(* CODESYS project lcls-twincat-motion-v1.3.3 (1).library
   Company: SLAC
   Title: lcls-twincat-motion
   Placeholder: lcls-twincat-motion
   Version: 1.3.3

Project tree, tasks and I/O mapping:
  libraries: LCLS General, * (SLAC); PMPS, * (SLAC - LCLS); Tc2_EtherCAT, * (Beckhoff Automation GmbH); Tc2_MC2, * (Beckhoff Automation GmbH); Tc2_Standard, * (Beckhoff Automation GmbH); Tc2_System, * (Beckhoff Automation GmbH); Tc2_Utilities, * (Beckhoff Automation GmbH); Tc3_Module, * (Beckhoff Automation GmbH)
  DUTs/
    data type DUT_MotionPneumaticActuator
    data type DUT_MotionStage
    data type DUT_PositionState
    data type EL5042_Status
    data type ENUM_EpicsHomeCmd
    data type ENUM_EpicsInOut
    data type ENUM_EpicsMotorCmd
    data type ENUM_MotionRequest
    data type ENUM_PnuematicActuatorPositionState
    data type ENUM_StageBrakeMode
    data type ENUM_StageEnableMode
    data type ST_RenishawAbsEnc
  GVLs/
    global variables MOTION_GVL
  POUs/
    Deprecated/
      function block FB_EpicsInOut [ST]
      function block FB_PositionStateManager [ST]
      function block FB_StatePTPMove [ST]
    ImplicitChecks/
      function CheckBounds [ST]
      function CheckDivDInt [ST]
      function CheckDivLInt [ST]
      function CheckDivLReal [ST]
      function CheckDivReal [ST]
    Motion/
      Gantry/
        function block FB_GantryAutoCoupling [ST]
        function block FB_GantryDiffVirtualLimitSwitch [ST]
      PMPS/
        function block FB_EncErrorFFO [ST]
        function block FB_NCErrorFFO [ST]
        function block FB_PositionStatePMPS [ST]: AssertHere, ClearAsserts, HandleBPTM, HandleFFO
        function block FB_PositionStatePMPS_Base [ST]: AssertHere, ClearAsserts, Exec, GetBeamFromState, GetStateCode, GetStateStruct, HandleBPTM, HandleFFO
        function block FB_PositionStatePMPS_Test [ST]: HandleBPTM, HandleFFO
      States/
        Examples/
          function block FB_PositionStateInOut [ST]
          function block FB_PositionStateInOut_WithPMPS [ST]
          function block FB_PositionStateInOut_WithPMPS_Test [ST]
        Helpers/
          function F_AtPositionState [ST]
          function F_PosOverLowerBound [ST]
          function F_PosUnderUpperBound [ST]
          function F_PosWithinDelta [ST]
          function block FB_RawCountConverter [ST]
        Internals/
          function block FB_PositionStateInternal [ST]
          function block FB_PositionStateLock [ST]
        function block FB_PositionStateBase [ST]: Exec, StateHandler
        function block FB_PositionStateBase_WithPMPS [ST]: Exec, PMPSHandler
        function block FB_PositionStateBase_WithPMPS_Test [ST]: Exec, PMPSHandler
        function block FB_PositionStateMove [ST]
      Utils/
        function F_MotionErrorCodeLookup [ST]
        function block FB_SetEnables [ST]
      function block FB_EncoderValue [ST]
      function block FB_MotionPneumaticActuator [ST]: ACT_IO, ACT_Logger
      function block FB_MotionRequest [ST]
      function block FB_MotionStage [ST]
      function block FB_MotionStageNCParams [ST]
      function block FB_MotionStageSim [ST]
    MotorTesting/
      function block FB_MicroStepCountTest [ST]
  tc_mca_std_lib/
    DUTs/
      data type DUT_AxisStatus_v0_01
    GVLs/
      global variables GVL
    POUs/
      ChangeConfig/
        function block FB_ReadFloatParameter [ST]
        function block FB_ReadParameterInNc_v1_00 [ST]
        function block FB_WriteFloatParameter [ST]
        function block FB_WriteParameterInNc_v1_00 [ST]
      ErrorHandling/
        data type DUT_ErrorState
        data type DUT_TerminalError
        function block FB_ErrorList [ST]
        function block FB_TerminalError [ST]
        global variables GVL_ErrorSystem
        data type ST_ErrorSystem
      Hardware/
        EtherCAT_Terminals/
          Analog_Inputs/
            function block EL3174_0002 [ST]
            function block EL3214 [ST]
            function block EL3255 [ST]
            function block FB_CalculateFrequency_3702_v0_01 [ST]
          Digital_Inputs/
            function block EL1008 [ST]
            function block EL1018 [ST]
            function block EL1808 [ST]
            function block EL1809 [ST]
            function block EL1819 [ST]
            function block FB_EL1252ASM_v1_00 [ST]
          Digital_Outputs/
            External_Types/
              data type dutEL2521_Ctrl
              data type dutEL2521_Status
            function block EL2014 [ST]
            function block EL2252 [ST]
            function block EL2808 [ST]
            function block EL2819 [ST]
          Measuring_Terminals/
            function block EL5002 [ST]
            function block EL5021 [ST]
            function block EL5042 [ST]
            function block EL5101 [ST]
          Motion/
            function block EL7211_v1_00 [ST]
            function block EL9576_v1_00 [ST]
          System/
            function block EL9410 [ST]
            function block EL9505 [ST]
        Other/
          function block EK1200 [ST]
      Motion/
        Homing/
          function block FB_HomeDirect [ST]
          function block FB_HomeFinish [ST]
          function block FB_HomePrepare [ST]
          function block FB_HomeReadNcVelocities [ST]
          function block FB_HomeReadSoftLimEnable [ST]
          function block FB_HomeToSwitch [ST]
          function block FB_HomeVirtual [ST]
          function block FB_HomeWriteNcVelocities [ST]
          function block FB_HomeWriteSoftLimEnable [ST]
        function block FB_DriveVirtual [ST]
        function block FB_NcAxis [ST]
  UnitTests/
    program BasicTests [ST]
    program Interactive [ST]
  Version/
    global variables Global_Version
*)

// DUTs/DUT_MotionPneumaticActuator
{attribute 'qualified_only'}
{attribute 'strict'}
TYPE DUT_MotionPneumaticActuator :
    // Defines the EPICS interface to actuating a pneumatic stage
STRUCT
     (* Hardware *)
    //Readbacks
    //Limit Switch
    {attribute 'pytmc' := '
     pv: PLC:bInLimitSwitch
     io: i
     field: ZNAM FALSE
     field: ONAM TRUE
     field: DESC TRUE if IN limit is reached
    '}
    i_bInLimitSwitch    :    BOOL;
    {attribute 'pytmc' := '
     pv: PLC:bOutLimitSwitch
     io: i
     field: ZNAM FALSE
     field: ONAM TRUE
     field: DESC TRUE if OUT limit is reached
    '}
    i_bOutLimitSwitch    :    BOOL;
    //Controls
    //Digital outputs
    {attribute 'pytmc' := '
    pv: bRetractDigitalOutput;
    io: i;
    field: ONAM FALSE
    field: ZNAM TRUE
    field: DESC TRUE if Retract digital output is active
    '}
    q_bRetract    :    BOOL;
    {attribute 'pytmc' := '
    pv: bInsetDigitalOutput;
    io: i;
    field: ONAM FALSE
    field: ZNAM TRUE
    field: DESC TRUE if Insert digital output is active
    '}
    q_bInsert    :    BOOL;


    //Logic and supervisory
    {attribute 'pytmc' := '
    pv: bInterlockOK;
    io: i;
    field: ZNAM FALSE
    field: ONAM TRUE
    field: DESC True if the actuator has permission to move in either direction
    '}
    bILK_OK: BOOL;
    {attribute 'pytmc' := '
    pv: bInsertEnable;
    io: i;
    field: ZNAM FALSE
    field: ONAM TRUE
    field: DESC True if the actuator had permission to be retracted
    '}
    bInsertOK    :    BOOL;
    {attribute 'pytmc' := '
    pv: bRetractEnable;
    io: i;
    field: ZNAM FALSE
    field: ONAM TRUE
    field: DESC True if the actuator had permission to be inserted
    '}
    bRetractOK    :    BOOL;

    (* Commands *)
    // Used from Epics to comand the actuator to  move
    {attribute 'pytmc' := '
    pv: CMD:IN;
    io: io;
    field: DESC Used by EPICS and internally to request Insert motion
    '}
    bInsert_SW        :    BOOL;
    {attribute 'pytmc' := '
    pv: CMD:OUT;
    io: io;
    field: DESC Used by EPICS and internally to request retract motion
    '}
    bRetract_SW    :    BOOL;

    (*Returns*)
     // TRUE if in the middle of a command
    {attribute 'pytmc' := '
     pv: bBusy
     io: i
     field: ONAM FALSE
     field: ZNAM TRUE
     field: DESC TRUE if in the middle of a command
    '}
    bBusy: BOOL;
    // TRUE if we've done a command and it has finished
    {attribute 'pytmc' := '
     pv: bDone
     io: i
     field: ONAM FALSE
     field: ZNAM TRUE
      field: DESC TRUE if command finished successfully
    '}
    bDone: BOOL;
     {attribute 'pytmc' := '
        pv: bReset
        io: io
        field: ZNAM FALSE
        field: ONAM TRUE
        field: DESC Used internally to reset errors
    '}
    bReset: BOOL;
    // TRUE if we're in an error state
    {attribute 'pytmc' := '
     pv: PLC:bError
     io: i
     field: ONAM FALSE
     field: ZNAM TRUE
     field: DESC TRUE if we're in an error state
    '}
    bError: BOOL;

     // Error code if nonzero
    {attribute 'pytmc' := '
     pv: PLC:nErrorId
     io: i
     field: DESC Error code if nonzero
    '}
    nErrorId: UDINT;
    // Message to identify the error state
    {attribute 'pytmc' := '
     pv: PLC:sErrorMessage
     io: i
     field: DESC Message to identify the error state
    '}
    sErrorMessage: STRING;
    {attribute 'pytmc' := '
    pv: nPositionState ;
    type: mbbi ;
    field: ZRST RETRACTED ;
    field: ONST INSERTED ;
    field: TWST MOVING ;
    field: THST INVALID ;
    io: i
    field: DESC Pneumatic actuator position
    '}

    eState    :    ENUM_PnuematicActuatorPositionState := ENUM_PnuematicActuatorPositionState.INVALID;

END_STRUCT
END_TYPE

// DUTs/DUT_MotionStage
TYPE DUT_MotionStage :
    // Defines the EPICS interface to moving a motor in TwinCAT
STRUCT
    (* Hardware *)

    // PLC Axis Reference
    Axis: AXIS_REF;
    // NC Forward Limit Switch: TRUE if ok to move
    {attribute 'pytmc' := '
        pv: PLC:bLimitForwardEnable
        io: i
        field: ZNAM FALSE
        field: ONAM TRUE
        field: DESC FALSE if forward limit hit
    '}
    bLimitForwardEnable AT %I*: BOOL;
    // NC Backward Limit Switch: TRUE if ok to move
    {attribute 'pytmc' := '
        pv: PLC:bLimitBackwardEnable
        io: i
        field: ZNAM FALSE
        field: ONAM TRUE
        field: DESC FALSE if reverse limit hit
    '}
    bLimitBackwardEnable AT %I*: BOOL;
    // NO Home Switch: TRUE if at home
    {attribute 'pytmc' := '
        pv: PLC:bHome
        io: i
        field: ZNAM FALSE
        field: ONAM TRUE
        field: DESC TRUE if at homing switch
    '}
    bHome AT %I*: BOOL;
    // NC Brake Output: TRUE to release brake
    {attribute 'pytmc' := '
        pv: PLC:bBrakeRelease
        io: i
        field: ZNAM FALSE
        field: ONAM TRUE
        field: DESC TRUE if brake released
    '}
    bBrakeRelease AT %Q*: BOOL;
    // NC STO Input: TRUE if ok to move
    {attribute 'pytmc' := '
        pv: PLC:bHardwareEnable
        io: i
        field: ZNAM FALSE
        field: ONAM TRUE
        field: DESC TRUE if STO not hit
    '}
    bHardwareEnable AT %I*: BOOL;

    // Raw encoder IO for ULINT (Biss-C)
    nRawEncoderULINT AT %I*: ULINT;
    // Raw encoder IO for UINT (Relative Encoders)
    nRawEncoderUINT AT %I*: UINT;
    // Raw encoder IO for INT (LVDT)
    nRawEncoderINT AT %I*: INT;

    (* Psuedo-hardware *)

    // Forward enable EPS summary
    {attribute 'pytmc' := '
        pv: PLC:bAllForwardEnable
        io: i
        field: ZNAM FALSE
        field: ONAM TRUE
        field: DESC Summary of axis permission to move forward
    '}
    bAllForwardEnable: BOOL:=FALSE;
    // Backward enable EPS summary
    {attribute 'pytmc' := '
        pv: PLC:bAllBackwardEnable
        io: i
        field: ZNAM FALSE
        field: ONAM TRUE
        field: DESC Summary of axis permission to move backward
    '}
    bAllBackwardEnable: BOOL:=FALSE;
    // Enable EPS summary encapsulating emergency stop button and any additional motion preventive hardware
    {attribute 'pytmc' := '
        pv: PLC:bAllEnable
        io: i
        field: ZNAM FALSE
        field: ONAM TRUE
        field: DESC Summary of axis permission to have power
    '}
    bAllEnable: BOOL:=FALSE;
    // Forward virtual gantry limit switch
    {attribute 'pytmc' := '
        pv: PLC:bGantryForwardEnable
        io: i
        field: ZNAM FALSE
        field: ONAM TRUE
        field: DESC TRUE if gantry ok to move forward
    '}
    bGantryForwardEnable: BOOL:=FALSE;
    // Backward virtual gantry limit switch
    {attribute 'pytmc' := '
        pv: PLC:bGantryBackwardEnable
        io: i
        field: ZNAM FALSE
        field: ONAM TRUE
        field: DESC TRUE if gantry ok to move backward
    '}
    bGantryBackwardEnable: BOOL:=FALSE;
    // Encoder count summary, if linked above
    {attribute 'pytmc' := '
        pv: PLC:nEncoderCount
        io: i
        field: DESC Count from encoder hardware
    '}
    nEncoderCount: UDINT;

    (* Settings *)
    // Name to use for log messages, fast faults, etc.
    {attribute 'pytmc' := '
        pv: PLC:sName
        io: i
        field: DESC PLC program name
    '}
    sName: STRING;
    // If TRUE, we want to enable the motor independently of PMPS or other safety systems.
    {attribute 'pytmc' := '
        pv: PLC:bPowerSelf
        io: i
        field: ZNAM FALSE
        field: ONAM TRUE
        field: DESC FALSE if axis is in PMPS
    '}
    bPowerSelf: BOOL:=FALSE;
    // Determines when we automatically enable the motor
    {attribute 'pytmc' := '
        pv: PLC:nEnableMode
        io: i
        field: DESC Describes when the axis will automatically get power
    '}
    nEnableMode: ENUM_StageEnableMode:=ENUM_StageEnableMode.DURING_MOTION;
    // Determines when we automatically disengage the brake
    {attribute 'pytmc' := '
        pv: PLC:nBrakeMode
        io: i
        field: DESC Describes when the brake will be released
    '}
    nBrakeMode: ENUM_StageBrakeMode:=ENUM_StageBrakeMode.IF_ENABLED;
    // Determines our encoder homing strategy
    {attribute 'pytmc' := '
        pv: PLC:nHomingMode
        io: i
        field: DESC Describes our homing strategy
    '}
    nHomingMode: ENUM_EpicsHomeCmd:=ENUM_EpicsHomeCmd.NONE;
    // Set true to activate gantry EPS
    {attribute 'pytmc' := '
        pv: PLC:bGantryAxis
        io: i
        field: ZNAM FALSE
        field: ONAM TRUE
        field: DESC TRUE if gantry EPS active
    '}
    bGantryAxis: BOOL:=FALSE;

    // Set to gantry difference tolerance
    nGantryTol: LINT:=0;

    // Encoder count at which this axis is aligned with other axis
    nEncRef: ULINT:=0;

    (* Commands *)
    // Used internally to request enables
    {attribute 'pytmc' := '
        pv: PLC:bEnable
        io: io
        field: ZNAM FALSE
        field: ONAM TRUE
        field: DESC Used internally to request enables
    '}
    bEnable: BOOL;
    // Used internally to reset errors and other state
    {attribute 'pytmc' := '
        pv: PLC:bReset
        io: io
        field: ZNAM FALSE
        field: ONAM TRUE
        field: DESC Used internally to reset errors
    '}
    bReset: BOOL;
    // Used internally and by the IOC to start or stop a move
    {attribute 'pytmc' := '
        pv: PLC:bExecute
        io: io
        field: ZNAM FALSE
        field: ONAM TRUE
        field: DESC Used internally and by the IOC to start or stop
    '}
    bExecute: BOOL;

    (* Command Args *)
    // Used internally and by the IOC to pick what kind of move to do
    {attribute 'pytmc' := '
        pv: PLC:nCommand
        io: io
        field: DESC Used internally and by the IOC to pick move type
    '}
    nCommand: INT;
    // Used internally and by the IOC to pass additional data to some commands
    {attribute 'pytmc' := '
        pv: PLC:nCmdData
        io: io
        field: DESC Used internally and by the IOC to pass extra args
    '}
    nCmdData: INT;
    // Used internally and by the IOC to pick a destination for the move
    {attribute 'pytmc' := '
        pv: PLC:fPosition
        io: io
        field: DESC Used internally and by the IOC as the set position
    '}
    fPosition: LREAL;
    // Used internally and by the IOC to pick a move velocity
    {attribute 'pytmc' := '
        pv: PLC:fVelocity
        io: io
        field: DESC Used internally and by the IOC to set velocity
    '}
    fVelocity: LREAL;
    // Used internally and by the IOC to pick a move acceleration
    {attribute 'pytmc' := '
        pv: PLC:fAcceleration
        io: io
        field: DESC Used internally and by the IOC to set acceleration
    '}
    fAcceleration: LREAL;
    // Used internally and by the IOC to pick a move deceleration
    {attribute 'pytmc' := '
        pv: PLC:fDeceleration
        io: io
        field: DESC Used internally and by the IOC to set deceleration
    '}
    fDeceleration: LREAL;
    // Used internally and by the IOC to pick a home position
    {attribute 'pytmc' := '
        pv: PLC:fHomePosition
        io: io
        field: DESC Used internally and by the IOC to pick home position
    '}
    fHomePosition: LREAL;

    (* Info *)
    // Unique ID assigned to each axis in the NC
    {attribute 'pytmc' := '
        pv: PLC:nMotionAxisID
        io: i
        field: DESC Unique ID assigned to each axis in the NC
    '}
    nMotionAxisID: UDINT:=0;

    (* Returns *)
    // TRUE if done enabling
    {attribute 'pytmc' := '
        pv: PLC:bEnableDone
        io: i
        field: ONAM FALSE
        field: ZNAM TRUE
        field: DESC TRUE if done enabling
    '}
    bEnableDone: BOOL;
    // TRUE if in the middle of a command
    {attribute 'pytmc' := '
        pv: PLC:bBusy
        io: i
        field: ONAM FALSE
        field: ZNAM TRUE
        field: DESC TRUE if in the middle of a command
    '}
    bBusy: BOOL;
    // TRUE if we've done a command and it has finished
    {attribute 'pytmc' := '
        pv: PLC:bDone
        io: i
        field: ONAM FALSE
        field: ZNAM TRUE
        field: DESC TRUE if command finished successfully
    '}
    bDone: BOOL;
    // TRUE if we have safety permission to move
    {attribute 'pytmc' := '
        pv: PLC:bSafetyReady
        io: i
        field: ONAM FALSE
        field: ZNAM TRUE
        field: DESC TRUE if safe to start a move
    '}
    bSafetyReady: BOOL;
    // TRUE if we're in an error state
    {attribute 'pytmc' := '
        pv: PLC:bError
        io: i
        field: ONAM FALSE
        field: ZNAM TRUE
        field: DESC TRUE if we're in an error state
    '}
    bError: BOOL;
    // Error code if nonzero
    {attribute 'pytmc' := '
        pv: PLC:nErrorId
        io: i
        field: DESC Error code if nonzero
    '}
    nErrorId: UDINT;
    // Message to identify the error state
    {attribute 'pytmc' := '
        pv: PLC:sErrorMessage
        io: i
        field: DESC Message to identify the error state
    '}
    sErrorMessage: STRING;
    // Internal hook for custom error messages
    sCustomErrorMessage: STRING;
    // MC_ReadParameterSet Output
    stAxisParameters: ST_AxisParameterSet;
    // True if we've updated stAxisParameters at least once
    bAxisParamsInit: BOOL;

    // Misc axis status information for the IOC
    stAxisStatus: DUT_AxisStatus_v0_01;
END_STRUCT
END_TYPE

// DUTs/DUT_PositionState
TYPE DUT_PositionState :
    // Defines settings and current safety status for moves to specific positions for an axis
STRUCT
    // Name as queried via the NAME PV in EPICS
    {attribute 'pytmc' := '
        pv: NAME
        io: input
        field: DESC Name of this position state
    '}
    sName: STRING := 'Invalid';

    // Position associated with this state
    {attribute 'pytmc' := '
        pv: SETPOINT
        io: io
        field: DESC Axis position associated with this state
    '}
    fPosition: LREAL;

    {attribute 'pytmc' := '
        pv: ENCODER
        io: i
        field: DESC Encoder count associated with this state
    '}
    nEncoderCount: UDINT;

    // Maximum allowable deviation from fPosition while at the state
    {attribute 'pytmc' := '
        pv: DELTA
        io: io
        field: DRVL 0.0
        field: DESC Max deviation from position at this state
    '}
    fDelta: LREAL;

    // Speed at which to move to this state
    {attribute 'pytmc' := '
        pv: VELO
        io: io
        field: DESC Speed at which to move to this state
    '}
    fVelocity: LREAL;

    // (optional) Acceleration to use for moves to this state
    {attribute 'pytmc' := '
        pv: ACCL
        io: io
        field: DESC Acceleration to use for moves to this state
    '}
    fAccel: LREAL;

    // (optional) Deceleration to use for moves to this state
    {attribute 'pytmc' := '
        pv: DCCL
        io: io
        field: DESC Deceleration to use for moves to this state
    '}
    fDecel: LREAL;

    // Safety parameter. This must be set to TRUE by the PLC program to allow moves to this state. This is expected to change as conditions change.
    {attribute 'pytmc' := '
        pv: MOVE_OK
        io: i
        field: ZNAM FALSE
        field: ONAM TRUE
        field: DESC TRUE if the move would be safe
    '}
    bMoveOk: BOOL;

    // Signifies to FB_PositionStateLock that this state should be immutable
    {attribute 'pytmc' := '
        pv: LOCKED
        io: i
        field: ZNAM FALSE
        field: ONAM TRUE
        field: DESC TRUE if state is immutable
    '}
    bLocked: BOOL;

    // Set this to TRUE when you make your state. This defaults to FALSE so that uninitialized states can never be moved to
    {attribute 'pytmc' := '
        pv: VALID
        io: i
        field: ZNAM FALSE
        field: ONAM TRUE
        field: DESC TRUE if this is a real state
    '}
    bValid: BOOL;

    // Set this to TRUE when you want to use the raw encoder counts to define the state
    bUseRawCounts: BOOL;

    // Is set to TRUE by FB_PositionStateInternal when called
    bUpdated: BOOL;

    // Beam parameters associated with this state
    stBeamParams: ST_BeamParams := PMPS_GVL.cst0RateBeam;

    // Transition ID associated with this state
    nRequestAssertionID: UDINT;
END_STRUCT
END_TYPE

// DUTs/EL5042_Status
TYPE EL5042_Status :
STRUCT
END_STRUCT
END_TYPE

// DUTs/ENUM_EpicsHomeCmd
{attribute 'qualified_only'}
{attribute 'strict'}
TYPE ENUM_EpicsHomeCmd :
    // Defines the valid options for homing in FB_MotionStage
(
    LOW_LIMIT := 1, // Low limit switch
    HIGH_LIMIT := 2, // High limit switch
    HOME_VIA_LOW := 3, // Home switch via low switch
    HOME_VIA_HIGH := 4, // Home switch via high switch
    ABSOLUTE_SET := 15, // Set here to be fHomePosition
    NONE := -1 // Do not home, ever
);
END_TYPE

// DUTs/ENUM_EpicsInOut
{attribute 'qualified_only'}
// Example EPICS states enum for use in FB_PositionStateManager
// Remove strict attribute for easier handling
TYPE ENUM_EpicsInOut :
(
    UNKNOWN := 0, // UNKNOWN must be in slot 0 or the FB breaks
    OUT := 1, // OUT at slot 1 is a convention
    IN := 2
);
END_TYPE

// DUTs/ENUM_EpicsMotorCmd
{attribute 'qualified_only'}
{attribute 'strict'}
TYPE ENUM_EpicsMotorCmd :
    // Defines valid EPICS commands for nCommand
(
    JOG := 0,
    MOVE_VELOCITY := 1,
    MOVE_RELATIVE := 2,
    MOVE_ABSOLUTE := 3,
    MOVE_MODULO := 4,
    HOME := 10,
    GEAR := 30
);
END_TYPE

// DUTs/ENUM_MotionRequest
{attribute 'qualified_only'}
{attribute 'strict'}
TYPE ENUM_MotionRequest :
    // Defines behavior options for when FB_MotionRequest is run during an active move from another source
(
    WAIT := 0,
    INTERRUPT := 1,
    ABORT := 2
);
END_TYPE

// DUTs/ENUM_PnuematicActuatorPositionState
{attribute 'qualified_only'}
{attribute 'strict'}
// Defines the positions for a pnuematic actuator
TYPE ENUM_PnuematicActuatorPositionState :
(
   RETRACTED    := 0, // Out limit switch is active
   INSERTED    := 1, // In limit switch is active
   MOVING    := 2, // Neither limit switches is Active
   INVALID :=3 // Invalid state
);
END_TYPE

// DUTs/ENUM_StageBrakeMode
{attribute 'qualified_only'}
{attribute 'strict'}
TYPE ENUM_StageBrakeMode :
    // Defines when to send the brake disengage signal in FB_MotionStage
(
    IF_ENABLED, // Disengage brake when the motor is enabled
    IF_MOVING, // Disengage brake when the motor is moving
    NO_BRAKE // Do not change the brake state in FB_MotionStage
);
END_TYPE

// DUTs/ENUM_StageEnableMode
{attribute 'qualified_only'}
{attribute 'strict'}
TYPE ENUM_StageEnableMode :
    // Define conditions when FB_MotionStage automatically sets bEnable
(
    ALWAYS, // Always set bEnable to TRUE
    NEVER,  // Only change bEnable on errors
    DURING_MOTION  // Enable before motion, disable after motion
);
END_TYPE

// DUTs/ST_RenishawAbsEnc
// Renishaw BiSS-C absolute encoder used with an EL5042
TYPE ST_RenishawAbsEnc :
STRUCT
    Count AT %I*: ULINT; // Connect to encoder "Position" input
    Status: EL5042_Status; // Status struct placeholder
    Ref: ULINT; // Encoder zero position (useful for aligned position with gantries)
END_STRUCT
END_TYPE

// tc_mca_std_lib/DUTs/DUT_AxisStatus_v0_01
TYPE DUT_AxisStatus_v0_01 :
STRUCT
	bEnable: BOOL;
	bReset: BOOL;
	bExecute: BOOL;
	nCommand: UINT;
	nCmdData: UINT;
	fVelocity: LREAL;
	fPosition: LREAL;
	fAcceleration: LREAL;
	fDeceleration: LREAL;
	bJogFwd: BOOL;
	bJogBwd: BOOL;
	bLimitFwd: BOOL;
	bLimitBwd: BOOL;
	fOverride: LREAL := 100;
	bHomeSensor: BOOL;
	bEnabled: BOOL;
	bError: BOOL;
	nErrorId: UDINT;
	fActVelocity: LREAL;
	fActPosition: LREAL;
	fActDiff: LREAL;
	bHomed:BOOL;
	bBusy:BOOL;
END_STRUCT
END_TYPE

// tc_mca_std_lib/POUs/ErrorHandling/DUT_ErrorState
{attribute 'qualified_only'}
{attribute 'strict'}
TYPE DUT_ErrorState :
(
	None,
	Active,
	Inactive,
	Acknowledged
);
END_TYPE

// tc_mca_std_lib/POUs/ErrorHandling/DUT_TerminalError
TYPE DUT_TerminalError :
STRUCT
	//Error system related
	iTerminalID : INT;					//ID of the terminal
	Error_ID : ULINT := 0;				//ID for the Error entry
	ErrorState : DUT_ErrorState;		//State of the error
	
	//Error related
	nDateTimeOn : ULINT;				//Date and time when the error occured. Raw data
	sDateTimeOn : STRING(24);			//Date and time when the error occured. Readable format
	nDateTimeOff : ULINT;				//Date and time when the error disapeared. Raw data
	sDateTimeOff : STRING(24);			//Date and time when the error disapeared. Readable format
	bWcState : BOOL;					//WcState variable of the terminal
	uiInfoDataState : UINT;				//InfoData.State variable of the terminal
	sErrorMessage : STRING (128);		//Error message corresponding to WcState and InfoData.State
	ErrorType : INT; 					//Error types (priorities) need to be developed
END_STRUCT
END_TYPE

// tc_mca_std_lib/POUs/ErrorHandling/ST_ErrorSystem
TYPE ST_ErrorSystem :
STRUCT
	//Array of error data. Size = cSizeOfErrorData in the GVL
	aErrorData : ARRAY [0..GVL_ErrorSystem.cSizeOfErrorData - 1] OF DUT_TerminalError;
	lNextErrorID : ULINT := 1;					//ErrorID for the next error entry
	nNoErrors : UINT;							//Number of errors in the list
	nNoOverflows : INT := 0;					//Number of overflows. How many error entries have been lost
END_STRUCT
END_TYPE

// tc_mca_std_lib/POUs/Hardware/EtherCAT_Terminals/Digital_Outputs/External_Types/dutEL2521_Ctrl
TYPE dutEL2521_Ctrl :
STRUCT
	///The control word (CW) is located in the output process image, and is transmitted from the controller to the terminal.
	///CW.0 FREQ_SEL 0bin / 1bin  Rapid change of the base frequency (only if the ramp function is inactive):
	///0bin = Base frequency 1 (object 8001:02)
	///1bin = Base frequency 2 (object 8001:03) 
	FREQ_SEL: BOOL;
	///CW.1 RAMP_DIS 1bin Operation of the ramp function is cancelled, in spite of object 8000:06 being active; if travel distance control is active, it is interrupted by this bit 
	RAMP_DIS: BOOL;
	///CW.2 GO_COUNTER 1bin  If travel distance control is active (object 8000:0A), then a pre-set counter value is approached when the bit is set 
	GO_COUNTER: BOOL;
	///CW.5 CNT_CLR 1bin The contents of the counter is cleared or set (object 8000:0B) by this bit. 
	///Any overflow or underflow bits that might be set are also cleared by this bit. 
	///The process can be edge triggered or level triggered (object 8000:05). 
	CNT_CLR: BOOL;
END_STRUCT
END_TYPE

// tc_mca_std_lib/POUs/Hardware/EtherCAT_Terminals/Digital_Outputs/External_Types/dutEL2521_Status
TYPE dutEL2521_Status :
STRUCT
	///The status word (SW) is located in the input process image, and is transmitted from the terminal to the controller.
	///SW.0 SEL_ACK/END_COUNTER 1bin  Confirms the change of base frequency. At activated travel distance control: target counter value reached 
	SEL_ACK: BOOL;
	///SW.1 RAMP_ACTIVE 1bin Ramp is currently being followed 
	RAMP_ACTIVE: BOOL;
	///SW.2 UNDERFLOW 1bin This bit is set if the 16-bit counter underflows (0 -> 65535). It is reset when the counter drops below two thirds of its measuring range (43690 -> 43689) or immediately an overflow occurs. 
	UNDERFLOW: BOOL;
	///SW.3 OVERFLOW 1bin This bit is set if the 16-bit counter overflows (65535 -> 0). It is reset when the counter exceeds one third of its measuring range (21845 -> 21846) or immediately an underflow occurs 
	OVERFLOW: BOOL;
	///SW.4 INPUT_T 1bin Status of INPUT_T 
	INPUT_T: BOOL;
	///SW.5 INPUT_Z 1bin Status of INPUT_Z 
	INPUT_Z: BOOL;
	///SW.6 ERROR 1bin General error bit, included with overflow/underflow 
	ERROR: BOOL;
END_STRUCT
END_TYPE

// GVLs/MOTION_GVL
{attribute 'qualified_only'}
VAR_GLOBAL
    stUnknownState: DUT_PositionState := (sName := 'Unknown');
    stInvalidState: DUT_PositionState;
END_VAR
VAR_GLOBAL CONSTANT
    // Allocated space for 6 states besides Unknown (16 including Unknown is the max for an EPICS MBBI)
    MAX_STATES: INT := 6;
END_VAR

// tc_mca_std_lib/GVLs/GVL
VAR_GLOBAL
	nHomingError:UDINT:=16#14D00;
END_VAR

// tc_mca_std_lib/POUs/ErrorHandling/GVL_ErrorSystem
{attribute 'qualified_only'}
VAR_GLOBAL CONSTANT
	cSizeOfErrorData : UINT := 128;
	
END_VAR

// Version/Global_Version
{attribute 'TcGenerated'}
// This function has been automatically generated from the project information.
VAR_GLOBAL CONSTANT
	{attribute 'const_non_replaced'}
	{attribute 'linkalways'}
	stLibVersion_lcls-twincat-motion : ST_LibVersion := (iMajor := 1, iMinor := 3, iBuild := 3, iRevision := 0, sVersion := '1.3.3');
END_VAR

// POUs/Deprecated/FB_EpicsInOut
FUNCTION_BLOCK FB_EpicsInOut
// Example usage of FB_PositionStateManager for a simple IN/OUT axis. See NOTE: comments.
// Also usable as a drop-in for these cases (no need to roll your own in/out)
VAR_IN_OUT
    // Motor to apply states to
    stMotionStage: DUT_MotionStage;
    // Information about the OUT position
    stOut: DUT_PositionState; // NOTE: Do not pragma these, let it happen in the manager.
    // Information about the IN parameter
    stIn: DUT_PositionState;
END_VAR
VAR_INPUT
    // If TRUE, the motor will be moved when enumSet is changed
    bEnable: BOOL;
    // When changed, sets the destination and starts a move
    {attribute 'pytmc' := '
        pv: SET
        io: io
    '}
    enumSet: ENUM_EpicsInOut; // NOTE: Please copy this pragma exactly on your enumSet
END_VAR
VAR_OUTPUT
    // If TRUE, we are in an error state
    bError: BOOL; // NOTE: do not pragma these, already has pragma in manager
    // Error code
    nErrorId: UDINT;
    // Message associated with bError = TRUE
    sErrorMessage: STRING;
    // If TRUE, we are currently moving between states
    bBusy: BOOL;
    // If TRUE, we asked for a move between states, it completed successfully, and there is no ongoing move
    bDone: BOOL;
    // The current state readback
    {attribute 'pytmc' := '
        pv: GET
        io: i
    '}
    enumGet: ENUM_EpicsInOut; // NOTE: Please copy this pragma exactly on your enumGet
END_VAR
VAR
    bInit: BOOL;
    arrStates: ARRAY[1..15] OF DUT_PositionState;

    {attribute 'pytmc' := '
        pv:
        io: io
    '}
    fbStateManager: FB_PositionStateManager; // NOTE: Please copy this pragma exactly to pick up the standard PVs
END_VAR

// Fist cycle setup
IF NOT bInit THEN
    stOut.sName := 'OUT';
    stIn.sName := 'IN';
    bInit := TRUE;
END_IF

// Stuff first two values of the 15 element array for the manager
arrStates[1] := stOut;
arrStates[2] := stIn;

// Call the function block every cycle
fbStateManager(
    stMotionStage := stMotionStage,
    arrStates := arrStates,
    setState := enumSet,
    bEnable := bEnable,
    bError => bError,
    nErrorId => nErrorId,
    sErrorMessage => sErrorMessage,
    bBusy => bBusy,
    bDone => bDone,
    getState => enumGet); // Cannot do this assignment if enumGet has attribute strict

END_FUNCTION_BLOCK

// POUs/Deprecated/FB_PositionStateManager
FUNCTION_BLOCK FB_PositionStateManager
(*
    Handles EPICS moves between multiple states for a single axis
    Should be wrapped inside a block with enums for states,
    see FB_EpicsInOut for an example.
*)
VAR_IN_OUT
    // Motor to move
    stMotionStage: DUT_MotionStage;

    // Allocated space for 15 states besides Unknown (16 is the max for an EPICS MBBI)
    {attribute 'pytmc' := '
        pv:
        io: io
        expand: %.2d
    '}
    arrStates: ARRAY[1..15] OF DUT_PositionState;

    // Corresponding arrStates index to move to, or 0 if no move selected
    setState: INT;
END_VAR
VAR_INPUT
    // If TRUE, start a move when setState transitions to a nonzero number
    bEnable: BOOL;
    // On rising edge, reset this FB
    {attribute 'pytmc' := '
        pv: RESET
        io: io
        field: ZNAM False
        field: ONAM True
    '}
    bReset: BOOL;
END_VAR
VAR_OUTPUT
    // If TRUE, there is an error
    {attribute 'pytmc' := '
        pv: ERR
        io: i
        field: ZNAM False
        field: ONAM True
    '}
    bError: BOOL;
    // Error ID
    {attribute 'pytmc' := '
        pv: ERRID
        io: i
    '}
    nErrorId: UDINT;
    // The error that caused bError to flip TRUE
    {attribute 'pytmc' := '
        pv: ERRMSG
        io: i
    '}
    sErrorMessage: STRING;
    // If TRUE, we are moving the motor
    {attribute 'pytmc' := '
        pv: BUSY
        io: i
        field: ZNAM False
        field: ONAM True
    '}
    bBusy: BOOL;
    // If TRUE, we are not moving the motor and the last move completed successfully
    {attribute 'pytmc' := '
        pv: DONE
        io: i
        field: ZNAM False
        field: ONAM True
    '}
    bDone: BOOL;

    // The current position we are trying to reach, or 0
    goalState: INT;
    // The readback position
    getState: INT;
END_VAR
VAR
    bInit: BOOL;
    stUnknown: DUT_PositionState;
    stGoal: DUT_PositionState;
    fbStateMove: FB_PositionStateMove;
    fbStateInternal: ARRAY[1..15] OF FB_PositionStateInternal;
    nIndex: INT;
    bNewGoal: BOOL;
    bInnerExec: BOOL;
    bInnerReset: BOOL;
    rtReset: R_TRIG;
    bMoveRequested: BOOL;
END_VAR

// Reset just goes through the first-cycle init again
rtReset(CLK:=bReset);
IF rtReset.Q THEN
    bInit := FALSE;
END_IF

// First-cycle init
IF NOT bInit THEN
    bError := FALSE;
    sErrorMessage := '';
    bBusy := FALSE;
    bDone := FALSE;
    bNewGoal := FALSE;
    bInnerExec := FALSE;
    bInnerReset := TRUE;
    setState := 0;
    goalState := 0;
END_IF

// All state internal handlers
FOR nIndex := 1 TO 15 DO
    IF arrStates[nIndex].bValid THEN
        fbStateInternal[nIndex](
            stMotionStage:=stMotionStage,
            stPositionState:=arrStates[nIndex]);
    END_IF
END_FOR

// Check where we are by going through all possible states.
// Note this favors the highest-number state that we're at, it's up to you to make your states mutually exclusive.
getState := 0;
FOR nIndex := 1 TO 15 DO
    IF F_AtPositionState(stMotionStage:=stMotionStage, stPositionState:=arrStates[nIndex]) THEN
        getState := nIndex;
    END_IF
END_FOR

// Use the changing set pv as a rising-edge trigger
IF setState <> goalState THEN
    goalState := setState;
    bNewGoal := TRUE;
END_IF

// Special move handling for error/enable state
IF bError OR NOT bEnable THEN
    bInnerExec := FALSE;
// Reset inner block this cycle if we were already moving but want a new move
ELSIF bInnerExec AND bNewGoal THEN
    bInnerExec := FALSE;
    bInnerReset := TRUE;
// If we hit this branch, we're starting a new move
ELSIF bNewGoal THEN
    bInnerExec := TRUE;
    bInnerReset := FALSE;
    bNewGoal := FALSE;
END_IF

// Pick the correct goal structure or Unknown
IF goalState = 0 THEN
    stGoal := stUnknown;
ELSE
    stGoal := arrStates[goalState];
END_IF

// Do the move
fbStateMove(
    stMotionStage := stMotionStage,
    stPositionState := stGoal,
    bExecute := bInnerExec,
    bReset := bInnerReset,
    enumMotionRequest := ENUM_MotionRequest.INTERRUPT,
    bBusy => bBusy);

// Only pass up bDone information if this FB is active
IF bInnerExec THEN
    bDone := fbStateMove.bDone;
END_IF

// Pick up any new errors, but don't override uncleared existing errors
IF NOT bError THEN
    bError := fbStateMove.bError;
    nErrorId := fbStateMove.nErrorId;
    sErrorMessage := fbStateMove.sErrorMessage;
END_IF

// Reset the setpoint and goal to 0 if we're not doing anything
// because FB is waiting for a change from 0 to "something"
bMoveRequested := bInnerExec AND NOT bDone;
IF NOT bError AND NOT bNewGoal AND NOT bMoveRequested THEN
    setState := 0;
    goalState := 0;
    bInnerExec := FALSE;
END_IF

// Bring inner reset back low at the end of the init cycle so that it can be triggered again later
IF NOT bInit THEN
    bInit := TRUE;
    bInnerReset := FALSE;
END_IF

END_FUNCTION_BLOCK

// POUs/Motion/States/Helpers/F_AtPositionState
FUNCTION F_AtPositionState : BOOL
    // Check if the motor is within the state bounds
VAR_INPUT
    stMotionStage: DUT_MotionStage;
    stPositionState: DUT_PositionState;
END_VAR

// If state is defined, we are within the delta, and we are either not moving or our destination is within the delta, we are at the state
F_AtPositionState := stPositionState.bValid AND stPositionState.bUpdated
                     AND F_PosWithinDelta(stMotionStage.stAxisStatus.fActPosition, stPositionState)
                     AND ((NOT stMotionStage.bExecute) OR F_PosWithinDelta(stMotionStage.fPosition, stPositionState));

END_FUNCTION

// POUs/Motion/States/Helpers/F_PosWithinDelta
FUNCTION F_PosWithinDelta : BOOL
VAR_INPUT
    fPosition: LREAL;
    stPositionState: DUT_PositionState;
END_VAR

F_PosWithinDelta := F_PosOverLowerBound(fPosition, stPositionState) AND
                    F_PosUnderUpperBound(fPosition, stPositionState);

END_FUNCTION

// POUs/Motion/States/Helpers/F_PosOverLowerBound
FUNCTION F_PosOverLowerBound : BOOL
VAR_INPUT
    fPosition: LREAL;
    stPositionState: DUT_PositionState;
END_VAR

F_PosOverLowerBound := fPosition > (stPositionState.fPosition - ABS(stPositionState.fDelta));

END_FUNCTION

// POUs/Motion/States/Helpers/F_PosUnderUpperBound
FUNCTION F_PosUnderUpperBound : BOOL
VAR_INPUT
    fPosition: LREAL;
    stPositionState: DUT_PositionState;
END_VAR

F_PosUnderUpperBound := fPosition < (stPositionState.fPosition + ABS(stPositionState.fDelta));

END_FUNCTION

// POUs/Motion/States/FB_PositionStateMove
FUNCTION_BLOCK FB_PositionStateMove
// Request a move to a particular state from an axis controlled via EPICS
// pytmc PVs here only exposed if using directly and not through FB_PositionStateManager
VAR_IN_OUT
    // Motor to move
    stMotionStage: DUT_MotionStage;

    // State to move to
    {attribute 'pytmc' := '
        pv:
    '}
    stPositionState: DUT_PositionState;
END_VAR
VAR_INPUT
    // Start move on rising edge, stop move on falling edge
    {attribute 'pytmc' := '
        pv: GO
        io: io
        field: ZNAM False
        field: ONAM True
    '}
    bExecute: BOOL;

    // Rising edge error reset
    {attribute 'pytmc' := '
        pv: RESET
        io: io
        field: ZNAM False
        field: ONAM True
    '}
    bReset: BOOL;

    // Define behavior for when a move is already active
    enumMotionRequest: ENUM_MotionRequest := ENUM_MotionRequest.WAIT;
END_VAR
VAR_OUTPUT
    // TRUE if the motor is at this state
    {attribute 'pytmc' := '
        pv: AT_STATE
        io: input
        field: ZNAM False
        field: ONAM True
    '}
    bAtState: BOOL;

    // TRUE if we have an error
    {attribute 'pytmc' := '
        pv: ERR
        io: input
        field: ZNAM False
        field: ONAM True
    '}
    bError: BOOL;

    // Error code
    {attribute 'pytmc' := '
        pv: ERRID
        io: input
    '}
    nErrorID: UDINT;

    // Error description
    {attribute 'pytmc' := '
        pv: ERRMSG
        io: input
    '}
    sErrorMessage: STRING;

    // TRUE if we are moving to a state
    {attribute 'pytmc' := '
        pv: BUSY
        io: input
        field: ZNAM False
        field: ONAM True
    '}
    bBusy: BOOL;

    // TRUE if we are note moving and we reached a state successfully on our last move
    {attribute 'pytmc' := '
        pv: DONE
        io: input
        field: ZNAM False
        field: ONAM True
    '}
    bDone: BOOL;
END_VAR
VAR
    fbMotionRequest: FB_MotionRequest;
    bAllowMove: BOOL;
END_VAR

// Veto the move for uninitialized and unsafe states
bAllowMove := stPositionState.bMoveOk AND stPositionState.bValid AND stPositionState.bUpdated;

// Do the move
fbMotionRequest(
    stMotionStage := stMotionStage,
    bExecute := bExecute AND bAllowMove,
    bReset := bReset,
    enumMotionRequest := enumMotionRequest,
    fPos := stPositionState.fPosition,
    fVel := stPositionState.fVelocity,
    fAcc := stPositionState.fAccel,
    fDec := stPositionState.fDecel,
    bError => bError,
    nErrorId => nErrorId,
    sErrorMessage => sErrorMessage,
    bBusy => bBusy,
    bDone => bDone);

// Inject custom error if we can't move because of bMoveOk or bValid
IF bExecute AND NOT bAllowMove THEN
    bError := TRUE;
    IF stPositionState.bValid THEN
        nErrorId := 16#7901;
    ELSE
        nErrorId := 16#7902;
    END_IF
    sErrorMessage := F_MotionErrorCodeLookup(nErrorId := nErrorID);
END_IF

// This can be useful if we're running this FB standalone for some reason
bAtState := F_AtPositionState(stMotionStage:=stMotionStage, stPositionState:=stPositionState);

END_FUNCTION_BLOCK

// POUs/Motion/Utils/F_MotionErrorCodeLookup
FUNCTION F_MotionErrorCodeLookup : STRING
VAR_INPUT
    nErrorId: UDINT;
END_VAR
VAR
    msg: STRING;
END_VAR

CASE nErrorId OF
    // Common NC errors
    16#4221: msg:='Requested set velocity is not allowed';
    16#4222: msg:='Requested set position is not allowed';
    16#4225: msg:='Drive not ready during axis start';
    16#4260: msg:='Drive disabled';
    16#4357: msg:='Negative limit hit';
    16#4358: msg:='Positive limit hit';
    16#4550: msg:='Stall: position lag monitoring error';
    16#4467: msg:='Encoder error: invalid actual position data';
    16#4B07: msg:='Timeout axis function block after 6 seconds';

    // Custom error definitions
    16#7900: msg:='Aborted move request with active move in progress';
    16#7901: msg:='Position state unsafe';
    16#7902: msg:='Position state invalid';

    // Fallbacks
    0: msg:='';
    ELSE
        msg:='Contact PCDS to add new message';
END_CASE
F_MotionErrorCodeLookup := msg;

END_FUNCTION

// POUs/Motion/FB_MotionRequest
FUNCTION_BLOCK FB_MotionRequest
(*
    Request a move from an axis controlled via EPICS using FB_MotionStage
    This exists to manage situations where different bits of code may need to move the same motor.
    With just the DUT_MotionStage/FB_MotionStage setup it is possible for two function blocks to
    fight with and interfere with each other and with the EPICS commands.
*)
VAR_IN_OUT
    // Motor to move
    stMotionStage: DUT_MotionStage;
END_VAR
VAR_INPUT
    // Start move on rising edge, stop move on falling edge
    bExecute: BOOL;
    // Reset errors on rising edge
    bReset: BOOL;
    // Define behavior for when the motor is already moving
    enumMotionRequest: ENUM_MotionRequest := ENUM_MotionRequest.WAIT;
    // Goal position
    fPos: LREAL;
    // Move velocity
    fVel: LREAL;
    // Optional acceleration
    fAcc: LREAL;
    // Optional deceleration
    fDec: LREAL;
END_VAR
VAR_OUTPUT
    // True if in error state
    bError: BOOL;
    // Error code
    nErrorId: UDINT;
    // What the error code means
    sErrorMessage: STRING;
    // If TRUE, we are moving the motor
    bBusy: BOOL;
    // If TRUE, we are not moving the motor and our most recent move was successful
    bDone: BOOL;
END_VAR
VAR
    rtExec: R_TRIG;
    ftExec: F_TRIG;
    rtReset: R_TRIG;
    ftBusy: F_TRIG;
    nState: UINT := 0;
    bMyMove: BOOL;
    bCausedError: BOOL;
END_VAR
// Define local constants for our state machine states
VAR CONSTANT
    INIT: UINT := 0;
    WAIT_EXEC: UINT := 1;
    PICK_REQUEST: UINT := 2;
    WAIT_OTHER_MOVE: UINT := 3;
    STOP_OTHER_MOVE: UINT := 4;
    START_MOVE: UINT := 5;
    WAIT_MY_MOVE: UINT := 6;
    STOP_MY_MOVE: UINT := 7;
    DONE_MOVING: UINT := 8;
    ERROR: UINT := 9;
END_VAR

rtExec(CLK:=bExecute);
ftExec(CLK:=bExecute);
rtReset(CLK:=bReset);

// Go back to INIT state on reset
IF rtReset.Q THEN
    nState := INIT;
    stMotionStage.bReset := TRUE;
END_IF
IF rtExec.Q OR ftExec.Q THEN
    bDone := FALSE;
END_IF

CASE nState OF
    // Start by setting everything to a known value
    INIT:
        nState := WAIT_EXEC;
        bError := FALSE;
        sErrorMessage := '';
        bDone := FALSE;
        bCausedError := FALSE;
    // Normal "waiting for move command" state
    WAIT_EXEC:
        bMyMove := FALSE;
        // Looking for a rising edge on bExecute
        IF rtExec.Q THEN
            bDone := FALSE;
            nState := PICK_REQUEST;
        END_IF
    // Decide how to handle the request
    PICK_REQUEST:
        IF stMotionStage.bBusy THEN
            CASE enumMotionRequest OF
                ENUM_MotionRequest.WAIT:
                    nState := WAIT_OTHER_MOVE;
                ENUM_MotionRequest.INTERRUPT:
                    nState := STOP_OTHER_MOVE;
                ENUM_MotionRequest.ABORT:
                    nState := ERROR;
                    bError := TRUE;
                    nErrorId := 16#7900;
            END_CASE
        ELSE
            nState := START_MOVE;
        END_IF
    // Watch the other move, then see if it's our turn
    WAIT_OTHER_MOVE:
        IF NOT stMotionStage.bBusy THEN
            // Try to pick request again next cycle once the move is over
            nState := PICK_REQUEST;
        END_IF
    // Interrupt the other move, then go to start ours
    STOP_OTHER_MOVE:
        stMotionStage.bExecute := FALSE;
        IF NOT stMotionStage.bBusy THEN
            nState := START_MOVE;
        END_IF
    // Set the correct values on DUT_MotionStage to start a new absolute move
    START_MOVE:
        bMyMove := TRUE;
        stMotionStage.bExecute := TRUE;
        stMotionStage.nCommand := ENUM_EpicsMotorCmd.MOVE_ABSOLUTE;
        stMotionStage.fPosition := fPos;
        stMotionStage.fVelocity := fVel;
        stMotionStage.fAcceleration := fAcc;
        stMotionStage.fDeceleration := fDec;
        nState := WAIT_MY_MOVE;
    // Watch our ongoing move, look for the move to end or requests to stop the move from this FB
    WAIT_MY_MOVE:
        ftBusy(CLK:=stMotionStage.bBusy);
        IF ftBusy.Q THEN
            nState := DONE_MOVING;
        END_IF
        // Implement stop on falling trigger
        IF ftExec.Q THEN
            nState := STOP_MY_MOVE;
        END_IF
    // Request a stop and wait for it to happen
    STOP_MY_MOVE:
        stMotionStage.bExecute := FALSE;
        IF NOT stMotionStage.bBusy THEN
            nState := DONE_MOVING;
        END_IF
    // Pick out the bDone state and return to waiting
    DONE_MOVING:
        bDone := stMotionStage.bDone;
        nState := WAIT_EXEC;
    // Lock us into the error state until the FB is reset
    ERROR:
        bMyMove := FALSE;
END_CASE

// Transition to the ERROR state if applicable
IF bMyMove AND stMotionStage.bError THEN
    nState := ERROR;
    bError := TRUE;
    nErrorId := stMotionStage.nErrorId;
    bCausedError := TRUE;
END_IF
sErrorMessage := F_MotionErrorCodeLookup(nErrorId := nErrorId);

CASE nState OF
INIT, WAIT_EXEC, ERROR:
    bBusy := FALSE;
ELSE
    bBusy := TRUE;
END_CASE

END_FUNCTION_BLOCK

// POUs/Motion/FB_MotionStage
FUNCTION_BLOCK FB_MotionStage
(*
    Default implementation for PLC behavior when motor IOC asks for a move
    This can be extended or replaced in your PLC project if you want
    non-default behavior to arise from the motor record processing
*)
VAR_IN_OUT
    stMotionStage: DUT_MotionStage;
END_VAR
VAR
    fbDriveVirtual: FB_DriveVirtual;
    bExecute: BOOL;
    bFwdHit: BOOL;
    bBwdHit: BOOL;
    ftExec: F_TRIG;
    rtExec: R_TRIG;
    rtUserExec: R_TRIG;
    rtTarget: R_TRIG;
    fbSetEnables: FB_SetEnables;
    bPosGoal: BOOL;
    bNegGoal: BOOL;
    fbEncoderValue: FB_EncoderValue;
    fbNCParams: FB_MotionStageNCParams;
    bNewMoveReq: BOOL;
    bPrepareDisable: BOOL;
END_VAR

// Start with an accurate status
stMotionStage.Axis.ReadStatus();

rtUserExec(CLK := stMotionStage.bExecute);
bNewMoveReq S= rtUserExec.Q;
bNewMoveReq R= NOT stMotionStage.bExecute;
bPrepareDisable R= bNewMoveReq;

bPosGoal := stMotionStage.stAxisStatus.fActPosition < stMotionStage.fPosition;
bNegGoal := stMotionStage.stAxisStatus.fActPosition > stMotionStage.fPosition;

// Moves are automatically allowed if no safety hooks. Otherwise, some other code will set this.
stMotionStage.bSafetyReady S= stMotionStage.bPowerSelf;

// Handle auto-enable timing
CASE stMotionStage.nEnableMode OF
    ENUM_StageEnableMode.ALWAYS:
        stMotionStage.bEnable := TRUE;
    ENUM_StageEnableMode.DURING_MOTION:
        IF bNewMoveReq THEN
            IF bPosGoal THEN
                IF stMotionStage.bAllForwardEnable THEN
                    stMotionStage.bEnable := stMotionStage.bSafetyReady;
                ELSIF NOT stMotionStage.bError THEN
                    // Not an error, just a warning
                    stMotionStage.sErrorMessage := 'Cannot move past positive limit.';
                    stMotionStage.bExecute := FALSE;
                END_IF
            ELSIF bNegGoal THEN
                IF stMotionStage.bAllBackwardEnable THEN
                    stMotionStage.bEnable := stMotionStage.bSafetyReady;
                ELSIF NOT stMotionStage.bError THEN
                    // Not an error, just a warning
                    stMotionStage.sErrorMessage := 'Cannot move past negative limit.';
                    stMotionStage.bExecute := FALSE;
                END_IF
            END_IF
            IF stMotionStage.bEnable OR stMotionStage.bError THEN
                bNewMoveReq := FALSE;
            END_IF
        END_IF
END_CASE

// Do not start the move until we have power and the safety system says it is OK
bExecute := stMotionStage.bExecute AND stMotionStage.bEnableDone AND stMotionStage.bSafetyReady;

IF bExecute AND NOT stMotionStage.bError THEN
    // Reset local warnings if things are going well
    stMotionStage.sErrorMessage := '';
END_IF

// Automatically fill the correct nCmdData for homing
IF stMotionStage.nCommand = ENUM_EpicsMotorCmd.HOME THEN
    stMotionStage.nCmdData := stMotionStage.nHomingMode;
END_IF

// Update all enable booleans
fbSetEnables(stMotionStage:=stMotionStage);

// No moves allowed in error states
IF stMotionStage.bError THEN
    bExecute := FALSE;
END_IF

// Handle standard commands using ESS's FB
fbDriveVirtual(En:=TRUE,
    bEnable:=stMotionStage.bAllEnable,
    bReset:=stMotionStage.bReset,
    bExecute:=bExecute,
    nCommand:=INT_TO_UINT(stMotionStage.nCommand),
    nCmdData:=INT_TO_UINT(stMotionStage.nCmdData),
    fVelocity:=stMotionStage.fVelocity,
    fPosition:=stMotionStage.fPosition,
    fAcceleration:=stMotionStage.fAcceleration,
    fDeceleration:=stMotionStage.fDeceleration,
    bLimitFwd:=stMotionStage.bAllForwardEnable,
    bLimitBwd:=stMotionStage.bAllBackwardEnable,
    bHomeSensor:=stMotionStage.bHome,
    fHomePosition:=stMotionStage.fHomePosition,
    bPowerSelf:=stMotionStage.bPowerSelf,
    nMotionAxisID=>stMotionStage.nMotionAxisID,
    Axis:=stMotionStage.Axis);

// Update status again after the move starts or stops
stMotionStage.Axis.ReadStatus();

// Check for a new error
IF NOT stMotionStage.bError THEN
    stMotionStage.bError := fbDriveVirtual.bError;
    stMotionStage.nErrorId := fbDriveVirtual.nErrorId;
END_IF

// Set the error message if we have one
IF stMotionStage.bError THEN
    // Hook if other code wants to inject a non-NC error
    IF stMotionStage.sCustomErrorMessage <> '' THEN
        stMotionStage.sErrorMessage := stMotionSTage.sCustomErrorMessage;
    ELSE
        stMotionStage.sErrorMessage := F_MotionErrorCodeLookup(nErrorId := stMotionStage.nErrorId);
    END_IF
END_IF

// When we start, set the busy/done appropriately
rtExec(CLK:=bExecute);
IF rtExec.Q THEN
    stMotionStage.bBusy := TRUE;
    stMotionStage.bDone := FALSE;
END_IF

// Force everything off in case of error
IF stMotionStage.bError THEN
    stMotionStage.bBusy := FALSE;
    stMotionStage.bDone := FALSE;
    stMotionStage.bEnable := FALSE;
END_IF

// Check the limits and cancel execution if appropriate. Without this block we have infinite error spam
bFwdHit := stMotionStage.Axis.Status.PositiveDirection AND NOT stMotionStage.bAllForwardEnable;
bBwdHit := stMotionStage.Axis.Status.NegativeDirection AND NOT stMotionStage.bAllBackwardEnable;
IF bFwdHit OR bBwdHit THEN
    stMotionStage.bExecute := FALSE;
END_IF

// Check done moving via fbDriveVirtual and from Target Position Monitoring. Must satisfy both conditions.
ftExec(CLK:=stMotionStage.bExecute);
rtTarget(CLK:=stMotionStage.Axis.Status.InTargetPosition AND fbDriveVirtual.bDone);
IF rtTarget.Q OR ftExec.Q THEN
    IF NOT stMotionStage.bDone THEN
        stMotionStage.bDone := TRUE;
        stMotionStage.bBusy := FALSE;
        IF NOT stMotionStage.Axis.Status.Error THEN
            bExecute := FALSE;
            stMotionStage.bExecute := FALSE;
        END_IF
    END_IF
END_IF

// Handle auto-disable timing
bPrepareDisable S= stMotionStage.nEnableMode = ENUM_StageEnableMode.DURING_MOTION AND ftExec.Q;
// Delay the disable until we reach standstill, else brake issues or other race conditions
IF bPrepareDisable AND stMotionStage.Axis.Status.MotionState = MC_AXISSTATE_STANDSTILL THEN
    bPrepareDisable := FALSE;
    stMotionStage.bEnable := FALSE;
END_IF

// Get a definitive bEnabled reading
CASE stMotionStage.Axis.Status.MotionState OF
    // We are not enabled if there is an issue
    MC_AXISSTATE_UNDEFINED, MC_AXISSTATE_DISABLED, MC_AXISSTATE_ERRORSTOP:
        stMotionStage.bEnableDone := FALSE;
    ELSE
        stMotionStage.bEnableDone := TRUE;
END_CASE

// Handle the brake. TRUE means brake disabled/released
IF stMotionStage.nBrakeMode <> ENUM_StageBrakeMode.NO_BRAKE THEN
    CASE stMotionStage.Axis.Status.MotionState OF
        MC_AXISSTATE_UNDEFINED,
        MC_AXISSTATE_DISABLED,
        MC_AXISSTATE_ERRORSTOP:
            stMotionStage.bBrakeRelease := FALSE;
        MC_AXISSTATE_STANDSTILL:
            IF stMotionStage.nBrakeMode = ENUM_StageBrakeMode.IF_MOVING THEN
                stMotionStage.bBrakeRelease := FALSE;
            ELSE
                stMotionStage.bBrakeRelease := TRUE;
            END_IF
        ELSE
            stMotionStage.bBrakeRelease := TRUE;
    END_CASE
END_IF

// Sync the epics status struct
stMotionStage.stAxisStatus := fbDriveVirtual.stAxisStatus;
stMotionStage.stAxisStatus.bEnabled := stMotionStage.bEnableDone;

// Reset everything when bReset is flagged
IF stMotionStage.bReset THEN
    stMotionStage.bEnable := FALSE;
    stMotionStage.bReset := FALSE;
    stMotionStage.bExecute := FALSE;
    stMotionStage.bError := FALSE;
    stMotionStage.nErrorId := 0;
    stMotionStage.sErrorMessage := '';
    stMotionStage.sCustomErrorMessage := '';
    bExecute := FALSE;
END_IF

// Ignore homing if we have the setting for it
// e.g. for pre-calibrated absolute encoders
IF stMotionStage.nHomingMode = ENUM_EpicsHomeCmd.NONE THEN
    stMotionStage.stAxisStatus.bHomed := TRUE;
END_IF

fbEncoderValue(stMotionStage:=stMotionStage);
fbNCParams(
    stMotionStage:=stMotionStage,
    bEnable:=TRUE,
    tRefreshDelay:=T#1s);

END_FUNCTION_BLOCK

// tc_mca_std_lib/POUs/Motion/FB_DriveVirtual
///#########################################################
///Function block to run a virtual drive with Nc
///	Library:		
///	Tc2_MC2.lib
///
///	Global Variables:
///	
///	Data types:
///	
///	External functions:
///
///###########################################################
FUNCTION_BLOCK FB_DriveVirtual
VAR
	sVersion: STRING:='1.0.3';	
END_VAR
VAR_INPUT
	En: BOOL;
	bEnable: BOOL;
	bReset: BOOL;
	bExecute: BOOL;
	/////	nCommandLocal...
	/////	0 = Jog
	/////	1 = MoveVelocity
	/////	2 = MoveRelative
	/////	3 = MoveAbsolut
	/////	4 = MoveModulo
	/////	10 = Homing
	/////	20 = SuperInp >>>ToBe
	/////	30 = Gear
	nCommand: UINT;
	nCmdData: UINT;
	fVelocity: LREAL;
	fPosition: LREAL;
	fAcceleration: LREAL;
	fDeceleration: LREAL;
	bJogFwd: BOOL;
	bJogBwd: BOOL;
	bLimitFwd: BOOL;
	bLimitBwd: BOOL;	
	fOverride: LREAL := 100;
	bHomeSensor: BOOL;
	fHomePosition:LREAL;
	nHomeRevOffset: UINT;
	MasterAxis: AXIS_REF;
	bPowerSelf: BOOL;
END_VAR
VAR_OUTPUT
	EnO: BOOL;
	bEnabled: BOOL;
	bBusy: BOOL;
	bDone: BOOL;
	bError: BOOL;
	bHomed: BOOL;
	nErrorId: UDINT;
	nMotionAxisID:UDINT:=0;  //Axis id in Motion (NC)
	Status: ST_AxisStatus;
	fActVelocity: LREAL;
	fActPosition: LREAL;
	fActDiff: LREAL;
    sErrorMessage:STRING;
END_VAR
VAR_IN_OUT
	Axis: AXIS_REF;
END_VAR
VAR	
	nCommandLocal: UINT;
	nCmdDataLocal: UINT;
	bFirstScan: BOOL := TRUE;
	fbReset: MC_Reset;
	fbPower: MC_Power;
	fbHalt: MC_Halt;
	fbJog: MC_Jog;
	fbMoveVelocity: MC_MoveVelocity;
	fbMoveRelative: MC_MoveRelative;
	fbMoveAbsolute: MC_MoveAbsolute;
	fbMoveModulo: MC_MoveModulo;	
	fbHomeVirtual:FB_HomeVirtual;
	fbGearInDyn: MC_GearInDyn;
	fbGearOut: MC_GearOut;
	fbExecuteRiseEdge: R_TRIG;
	stAxisStatus: DUT_AxisStatus_v0_01;	
END_VAR

EnO:=En;

// Transfer nCommand and nCmdData to local copies at rising edge of bExecute (avoid issues if nCommand or nCmdData are changed during a command) 
fbExecuteRiseEdge(CLK:=bExecute);
IF fbExecuteRiseEdge.Q THEN
  nCmdDataLocal:=nCmdData;
  nCommandLocal:=nCommand;
END_IF

bHomed:=fbHomeVirtual.bHomed; //Add in DUT_AxisStatus later
bDone:=FALSE;

(*Reset*)
fbReset(
	Execute:=bReset AND Axis.Status.Error,
	Axis:=Axis,
	Done=> ,
	Busy=> ,
	Error=> ,
	ErrorID=> );

(*Power*)
IF bPowerSelf THEN
fbPower(
	Axis:=Axis,
	Enable:=bEnable,	
	Enable_Positive:=bEnable AND bLimitFwd,	
	Enable_Negative:=bEnable AND bLimitBwd,	
	Override:=fOverride,
	BufferMode:= ,
	Status=> ,
	Busy=> ,
	Active=> ,
	Error=> ,
	ErrorID=> );
END_IF

(*Halt*)
fbHalt(
	Execute:=NOT bExecute  AND (((fbMoveVelocity.Busy OR fbPower.Busy) AND (nCommandLocal=1)) OR (fbMoveRelative.Busy AND (nCommandLocal=2)) OR (fbMoveAbsolute.Busy AND (nCommandLocal=3)) OR (fbMoveModulo.Busy AND (nCommandLocal=4)) OR (fbHomeVirtual.bBusy AND (nCommandLocal=10))),
	Deceleration:=fDeceleration,
	Jerk:=0,
	BufferMode:= ,
	Options:= ,
	Axis:=Axis ,
	Done=> ,
	Busy=> ,
	Active=> ,
	CommandAborted=> ,
	Error=> ,
	ErrorID=> );

(*Jog (Command = 0)*)
fbJog(
	JogForward:=bJogFwd AND (nCommandLocal=0) ,
	JogBackwards:=bJogBwd AND (nCommandLocal=0) ,
	Mode:=UINT_TO_INT(nCmdDataLocal),
	Position:= ,
	Velocity:=fVelocity,
	Acceleration:=fAcceleration,
	Deceleration:=fDeceleration,
	Jerk:=0,
	Axis:=Axis,
	Done=> ,
	Busy=> ,
	Active=> ,
	CommandAborted=> ,
	Error=> ,
	ErrorID=> );

(*MoveVelocity (Command = 1)*)
fbMoveVelocity(
	Execute:=bExecute AND (nCommandLocal=1),
	Velocity:=ABS(fVelocity),
	Acceleration:=fAcceleration,
	Deceleration:=fDeceleration,
	Jerk:=0,
	Direction:=SEL(fVelocity<0, MC_Positive_Direction, MC_Negative_Direction),
	BufferMode:= ,
	Options:= ,
	Axis:=Axis,
	InVelocity=> ,
	Busy=> ,
	Active=> ,
	CommandAborted=> ,
	Error=> ,
	ErrorID=> );

(*MoveRelative (Command = 2)*)
fbMoveRelative(
	Execute:=bExecute AND (nCommandLocal=2), 
	Distance:=fPosition, 
	Velocity:=ABS(fVelocity), 
	Acceleration:=fAcceleration,
	Deceleration:=fDeceleration,
	Jerk:=0,
	BufferMode:= , 
	Options:= , 
	Axis:=Axis, 
	Done=> , 
	Busy=> , 
	Active=> , 
	CommandAborted=> , 
	Error=> , 
	ErrorID=> );
	
IF nCommandLocal=2 THEN
	bDone:=fbMoveRelative.Done;
END_IF
	
(*MoveAbsolute (Command = 3)*)
fbMoveAbsolute(
	Execute:=bExecute AND (nCommandLocal=3),
	Position:=fPosition,
	Velocity:=ABS(fVelocity),
	Acceleration:=fAcceleration,
	Deceleration:=fDeceleration,
	Jerk:=0,
	BufferMode:= ,
	Options:= ,
	Axis:=Axis,
	Done=> ,
	Busy=> ,
	Active=> ,
	CommandAborted=> ,
	Error=> ,
	ErrorID=> );

IF nCommandLocal=3 THEN
	bDone:=fbMoveAbsolute.Done;
END_IF

(*MoveModulo (Command = 4)*)
fbMoveModulo(
	Execute:=bExecute AND (nCommandLocal=4), 
	Position:=fPosition, 
	Velocity:=ABS(fVelocity), 
	Acceleration:=fAcceleration, 
	Deceleration:=fDeceleration, 
	Jerk:=0, 
	Direction:=UINT_TO_INT(nCmdDataLocal), 
	BufferMode:= , 
	Options:= , 
	Axis:=Axis, 
	Done=> , 
	Busy=> , 
	Active=> , 
	CommandAborted=> , 
	Error=> , 
	ErrorID=> );

IF nCommandLocal=4 THEN
	bDone:=fbMoveModulo.Done;
END_IF
	
(*Home (Command = 10)*)
fbHomeVirtual(	
	bExecute:= nCommandLocal=10 AND bExecute,
	fHomePosition:=fHomePosition,
	bHomeSensor:=bHomeSensor,
	bLimitBwd:=bLimitBwd,
	bLimitFwd:=bLimitFwd,
	nCmdData:=nCmdDataLocal,
	bReset:=bReset,
	nHomeRevOffset:=nHomeRevOffset,
	Axis:=Axis
	);
	
IF nCommandLocal=10 THEN
	bDone:=fbHomeVirtual.bDone;
END_IF
	
(*Gear (Command = 30)*)
fbGearInDyn(
	Enable:=bExecute  AND (nCommandLocal=30),
	GearRatio:=SEL(nCmdDataLocal>0, 1,fVelocity),
	Acceleration:=fAcceleration,
	Deceleration:=fDeceleration,
	Jerk:=0.0,
	BufferMode:= , 
	Options:= , 
	Master:=MasterAxis,
	Slave:=Axis,
	InGear=> , 
	Busy=> , 
	Active=> , 
	CommandAborted=> , 
	Error=> , 
	ErrorID=> );
	
fbGearOut(
	Execute:=NOT bExecute AND Axis.Status.NotMoving AND (nCommandLocal=30),
	Slave:=Axis,
	Error=>,
	Done=>,
	ErrorID=>);


IF nCommandLocal=30 THEN
	bDone:=Axis.Status.Coupled;
END_IF

(*Busy*)
bBusy:=Axis.Status.HasJob OR Axis.Status.HomingBusy OR fbHomeVirtual.bBusy;

(*Enabled*)
bEnabled:=fbPower.Status;

(*Error from functions and Nc*)
IF fbPower.Error AND fbPower.Active THEN
	bError:=fbPower.Enable;
	nErrorId:=fbPower.ErrorID;
ELSIF fbHalt.Error AND fbHalt.Active THEN
	bError:=fbHalt.Execute;
	nErrorId:=fbHalt.ErrorID;
ELSIF fbJog.Error AND nCommandLocal=0 (*fbJog.Active*) THEN
	bError:=fbJog.JogForward OR fbJog.JogBackwards;
	nErrorId:=fbJog.ErrorID;
ELSIF fbMoveVelocity.Error AND nCommandLocal=1(*fbMoveVelocity.Active*) THEN
	bError:=fbMoveVelocity.Execute;
	nErrorId:=fbMoveVelocity.ErrorID;
ELSIF fbMoveRelative.Error AND nCommandLocal=2 (*fbMoveRelative.Active*) THEN
	bError:=fbMoveRelative.Execute;
	nErrorId:=fbMoveRelative.ErrorID;
ELSIF fbMoveAbsolute.Error AND nCommandLocal=3 (*fbMoveAbsolute.Active*) THEN
	bError:=fbMoveAbsolute.Execute;
	nErrorId:=fbMoveAbsolute.ErrorID;
ELSIF fbMoveModulo.Error AND nCommandLocal=4 (*fbMoveModulo.Active*) THEN
	bError:=fbMoveModulo.Execute;
	nErrorId:=fbMoveModulo.ErrorID;
ELSIF fbHomeVirtual.bError AND nCommandLocal=10 (*fbHome.Active*) THEN
	bError:=fbHomeVirtual.bError;
	nErrorId:=fbHomeVirtual.nErrorID;
ELSIF fbGearInDyn.Error AND nCommandLocal=30 (*fbGearInDyn.Active*) THEN
	bError:=fbGearInDyn.Enable;
	nErrorId:=fbGearInDyn.ErrorID;
ELSIF fbGearOut.Error AND nCommandLocal=30 AND Axis.Status.Coupled THEN
	bError:=fbGearOut.Execute;
	nErrorId:=fbGearOut.ErrorID;
ELSIF Axis.Status.Error  THEN
	bError:=TRUE;
	nErrorId:=Axis.Status.ErrorID;
ELSIF fbHomeVirtual.bError THEN
	bError:=TRUE;
	nErrorId:=fbHomeVirtual.nErrorId;
ELSE
	bError:=FALSE;
	nErrorId:=0;
END_IF;

(*Converese nErrorID to string*)
sErrorMessage:=WORD_TO_HEXSTR(in:=TO_WORD(nErrorID) , iPrecision:= 4, bLoCase:=0 );

(*Status from Nc*)
Status:=Axis.Status;

(*Axis id in motion "motor"*)
nMotionAxisID:=axis.NcToPlc.AxisId;

(*Actual Velocity*)
fActVelocity:=Axis.NcToPlc.ActVelo;

(*Actual Position*)
IF Axis.Status.OpMode.Modulo THEN
	fActPosition:=Axis.NcToPlc.ModuloActPos;
ELSE
	fActPosition:=Axis.NcToPlc.ActPos;
END_IF

(*Actual Position*)
fActDiff:=Axis.NcToPlc.PosDiff;


//Status struct for EPICS communication
stAxisStatus.bEnable:=bEnable;
stAxisStatus.bEnabled:=bEnabled;
stAxisStatus.bError:=bError;
stAxisStatus.bExecute:=bExecute;
stAxisStatus.bHomeSensor:=bHomeSensor;
stAxisStatus.bJogBwd:=bJogBwd;
stAxisStatus.bJogFwd:=bJogFwd;
stAxisStatus.bLimitBwd:=bLimitBwd;
stAxisStatus.bLimitFwd:=bLimitFwd;
stAxisStatus.bReset:=bReset;
stAxisStatus.fAcceleration:=fAcceleration;
stAxisStatus.fActDiff:=fActDiff;
stAxisStatus.fActPosition:=fActPosition;
stAxisStatus.fActVelocity:=fActVelocity;
stAxisStatus.fDeceleration:=fDeceleration;
stAxisStatus.fOverride:=fOverride;
stAxisStatus.fPosition:=fPosition;
stAxisStatus.fVelocity:=fVelocity;
stAxisStatus.nCmdData:=nCmdData;  //Or nCmdDataLocal
stAxisStatus.nCommand:=nCommand;  //Or nCommandLocal
stAxisStatus.nErrorId:=nErrorId;
stAxisStatus.bBusy:=bBusy;
stAxisStatus.bHomed:=bHomed;

IF bFirstScan THEN
	bFirstScan:=FALSE;
END_IF

END_FUNCTION_BLOCK

// tc_mca_std_lib/POUs/Motion/Homing/FB_HomeVirtual
FUNCTION_BLOCK FB_HomeVirtual
VAR_INPUT
	En: BOOL;
	bReset: BOOL;
	bExecute: BOOL;
	nCmdData: UINT;
	bLimitFwd: BOOL;
	bLimitBwd: BOOL;	
	bHomeSensor: BOOL;	
	fHomePosition:LREAL;
	nHomeRevOffset: UINT;
END_VAR
VAR_IN_OUT
	Axis: AXIS_REF;
END_VAR
VAR_OUTPUT
	EnO: BOOL;	
	bBusy: BOOL;
	bDone: BOOL;
	bHomed:BOOL;
	bError: BOOL;
	nErrorId: UDINT;
END_VAR
VAR
	fbHomeToSwitch: FB_HomeToSwitch;
    fbHomeDirect: FB_HomeDirect; //Only used for direct homing (set of position)
    fbMoveVelocity:MC_MoveVelocity;
    fbHomePrepare:FB_HomePrepare;
	fbHomeFinish:FB_HomeFinish;    	    		
	fbExecuteRiseEdge: R_TRIG;
    nHomingState:INT:=0;
	bExecuteHomeToSwitch:BOOL:=FALSE;
	bExecuteMoveVelocity:BOOL:=FALSE;
	bExecutePrepare: BOOL:=FALSE;
	bExecuteFinish: BOOL:=FALSE;
	bExecuteHomeDirect: BOOL;
	nCmdDataLocal: UINT;  //Ensure that nCmdData is not changed during sequence
	bSequenceReady:BOOL:=TRUE;
	bRestoreNCDataNeeded: BOOL:=FALSE;
END_VAR

EnO:=En;

IF bReset THEN	
	bError:=FALSE;
	nErrorId:=0;
END_IF

// Reset when bExecute is low
IF NOT bExecute THEN
  nHomingState:=0;
  bSequenceReady:=TRUE;
  bExecuteHomeToSwitch:=FALSE;
  bExecuteHomeDirect:=FALSE;
  bExecuteMoveVelocity:=FALSE;
  bExecutePrepare:=FALSE;
  bExecuteFinish:=FALSE;
END_IF

//Reset at rinsing edge of bExecute
fbExecuteRiseEdge(CLK:=bExecute);
IF fbExecuteRiseEdge.Q THEN
  nCmdDataLocal:=nCmdData; //Ensure that nCmdData is not changed during sequence (nCmdData will only be read at a rising edge of bExecute)
  bSequenceReady:=FALSE;
  bExecutePrepare:=TRUE;  
  bRestoreNCDataNeeded:=FALSE;
  //Check if valid nCmdDataLocal
  CASE nCmdDataLocal OF  	
    1:
    2:
    3:
    4:
    15:
    ELSE //nCmdData not valid	
      bError:=TRUE;
      nErrorId:=16#4FFF;   
  END_CASE
END_IF

//############# Prepare for homing (Read from NC and reset homed flag)
fbHomePrepare(
  En:=En,
  bExecute:=bExecutePrepare AND NOT bError, // Not needed for sequence 15 (set position only, no movement))
  bReset:=bReset,
  Axis:=Axis,
);

//############# Homing Sequences:
CASE nCmdDataLocal OF  
	
   1: // Home to low limit switch
	   CASE nHomingState OF
		  0:
		    bHomed:=Axis.Status.Homed;
            // Wait for read of velocities from NC and reset of calibration flag
	        IF fbHomePrepare.bDone AND bExecute AND NOT bSequenceReady THEN
			  bRestoreNCDataNeeded:=TRUE;
			  IF bLimitBwd THEN
                nHomingState:=1;
              ELSE
				nHomingState:=2;  //Standing on limit switch go direct to state 2 
              END_IF                                          		  
	        END_IF
		  1: // wait for reach low limit then trigger fbHomeToSwitch
		    bHomed:=FALSE;
			bSequenceReady:=FALSE;
			fbMoveVelocity.Velocity:=ABS(fbHomePrepare.fVelocityToCam);
            fbMoveVelocity.Direction:=MC_Negative_Direction;
	        bExecuteMoveVelocity:=bExecute;  // Execute MC_MoveVelocity
		    IF NOT bLimitBwd AND NOT fbMoveVelocity.Busy AND Axis.Status.NotMoving THEN //MC_MoveVelocity.Busy goes down when ramp down initiates (not ends).
			  nHomingState:=2;
		    END_IF
		  2: // Wait for fbHomeToSwitch
		    bHomed:=FALSE;
		    bSequenceReady:=FALSE;
            bExecuteMoveVelocity:=FALSE;			
            bExecuteHomeToSwitch:=TRUE;	
            fbHomeToSwitch.nSearchDirTwoardsCam:=MC_Positive_Direction;
            fbHomeToSwitch.nSearchDirOffCam:=MC_Positive_Direction;	             
	        fbHomeToSwitch.fVelocityToCamNC:=fbHomePrepare.fVelocityToCam; // High speed
  	        fbHomeToSwitch.fVelocityFromCamNC:=fbHomePrepare.fVelocityFromCam;  // Low speed              		
		    fbHomeToSwitch.bCamSensor:=NOT bLimitBwd;            	 		    
	        IF fbHomeToSwitch.bDone THEN	          
			  nHomingState:=3;
			  bExecuteFinish:=TRUE;
			  fbHomeFinish.bSofLimEnableHigh:=fbHomePrepare.bSofLimEnableHighOriginal;
			  fbHomeFinish.bSofLimEnableLow:=fbHomePrepare.bSofLimEnableLowOriginal;
	        END_IF;	
          3: // restore softlimit enable
            bHomed:=FALSE;
		    bSequenceReady:=FALSE;            		            	
	        IF fbHomeFinish.bDone THEN
			  bRestoreNCDataNeeded:=FALSE;
	          bSequenceReady:=TRUE;
			  nHomingState:=0;
			  bHomed:=Axis.Status.Homed;
	        END_IF;	 
	   END_CASE;
	   
   2: // Home to high limit switch
	   CASE nHomingState OF
		  0:
		    bHomed:=Axis.Status.Homed;
            // Wait for read of velocities from NC and reset of calibration flag
	        IF fbHomePrepare.bDone AND bExecute AND NOT bSequenceReady THEN
			  bRestoreNCDataNeeded:=TRUE;
			  IF bLimitFwd THEN
                nHomingState:=1;
              ELSE
				nHomingState:=2;  //Standing on limit switch go direct to state 2 
              END_IF                                          		  
	        END_IF
		  1: // wait for reach low limit then trigger fbHomeToSwitch
		    bHomed:=FALSE;
			bSequenceReady:=FALSE;
			fbMoveVelocity.Velocity:=ABS(fbHomePrepare.fVelocityToCam);
            fbMoveVelocity.Direction:=MC_Positive_Direction;
	        bExecuteMoveVelocity:=bExecute;  // Execute MC_MoveVelocity
		    IF NOT bLimitFwd AND NOT fbMoveVelocity.Busy AND Axis.Status.NotMoving THEN //MC_MoveVelocity.Busy goes down when ramp down initiates (not ends).
			  nHomingState:=2;
		    END_IF
		  2: // Wait for fbHomeToSwitch
		    bHomed:=FALSE;
		    bSequenceReady:=FALSE;
            bExecuteMoveVelocity:=FALSE;			
            bExecuteHomeToSwitch:=TRUE;	
            fbHomeToSwitch.nSearchDirTwoardsCam:=MC_Negative_Direction;
            fbHomeToSwitch.nSearchDirOffCam:=MC_Negative_Direction;	             
	        fbHomeToSwitch.fVelocityToCamNC:=fbHomePrepare.fVelocityToCam; // High speed
  	        fbHomeToSwitch.fVelocityFromCamNC:=fbHomePrepare.fVelocityFromCam;  // Low speed              		
		    fbHomeToSwitch.bCamSensor:=NOT bLimitFwd;            	 		    
	        IF fbHomeToSwitch.bDone THEN	          
			  nHomingState:=3;
			  bExecuteFinish:=TRUE;
			  fbHomeFinish.bSofLimEnableHigh:=fbHomePrepare.bSofLimEnableHighOriginal;
			  fbHomeFinish.bSofLimEnableLow:=fbHomePrepare.bSofLimEnableLowOriginal;
	        END_IF;	
          3: // restore softlimit enable
            bHomed:=FALSE;
		    bSequenceReady:=FALSE;            		            	
	        IF fbHomeFinish.bDone THEN
			  bRestoreNCDataNeeded:=FALSE;
	          bSequenceReady:=TRUE;
			  nHomingState:=0;
			  bHomed:=Axis.Status.Homed;
	        END_IF;	 
	   END_CASE;
	   
   3: // Home on bHomeSensor via bLimitBwd
   	   CASE nHomingState OF
		  0:
		    bHomed:=Axis.Status.Homed;
            // Wait for read of velocities from NC and reset of calibration flag
	        IF fbHomePrepare.bDone AND bExecute AND NOT bSequenceReady THEN
			  bRestoreNCDataNeeded:=TRUE;
			  IF bLimitBwd THEN
                nHomingState:=1;
              ELSE
				nHomingState:=2;  //Standing on limit switch go direct to state 2 
              END_IF                                          		  
	        END_IF
		  1: // wait for reach low limit then trigger fbHomeToSwitch
		    bHomed:=FALSE;
			bSequenceReady:=FALSE;
			fbMoveVelocity.Velocity:=ABS(fbHomePrepare.fVelocityToCam);
            fbMoveVelocity.Direction:=MC_Negative_Direction;
	        bExecuteMoveVelocity:=bExecute;  // Execute MC_MoveVelocity
		    IF NOT bLimitBwd AND NOT fbMoveVelocity.Busy AND Axis.Status.NotMoving THEN //MC_MoveVelocity.Busy goes down when ramp down initiates (not ends).
			  nHomingState:=2;
		    END_IF
		  2: // Wait for fbHomeToSwitch
		    bHomed:=FALSE;
		    bSequenceReady:=FALSE;
            bExecuteMoveVelocity:=FALSE;			
            bExecuteHomeToSwitch:=TRUE;	
            fbHomeToSwitch.nSearchDirTwoardsCam:=MC_Positive_Direction;
            fbHomeToSwitch.nSearchDirOffCam:=MC_Positive_Direction;	             
	        fbHomeToSwitch.fVelocityToCamNC:=fbHomePrepare.fVelocityToCam; // High speed
  	        fbHomeToSwitch.fVelocityFromCamNC:=fbHomePrepare.fVelocityFromCam;  // Low speed              		
		    fbHomeToSwitch.bCamSensor:=bHomeSensor;            	 		    
	        IF fbHomeToSwitch.bDone THEN	          
			  nHomingState:=3;
			  bExecuteFinish:=TRUE;
			  fbHomeFinish.bSofLimEnableHigh:=fbHomePrepare.bSofLimEnableHighOriginal;
			  fbHomeFinish.bSofLimEnableLow:=fbHomePrepare.bSofLimEnableLowOriginal;
	        END_IF;	
          3: // restore softlimit enable
            bHomed:=FALSE;
		    bSequenceReady:=FALSE;            		            	
	        IF fbHomeFinish.bDone THEN
		      bRestoreNCDataNeeded:=FALSE;
	          bSequenceReady:=TRUE;
			  nHomingState:=0;
			  bHomed:=Axis.Status.Homed;
	        END_IF;	 
	   END_CASE;
	4:  // Home on bHomeSensor via bLimitFwd	   
	   CASE nHomingState OF
		  0:
		    bHomed:=Axis.Status.Homed;
            // Wait for read of velocities from NC and reset of calibration flag
	        IF fbHomePrepare.bDone AND bExecute AND NOT bSequenceReady THEN
			  bRestoreNCDataNeeded:=TRUE;
			  IF bLimitFwd THEN
                nHomingState:=1;
              ELSE
				nHomingState:=2;  //Standing on limit switch go direct to state 2 
              END_IF                                          		  
	        END_IF
		  1: // wait for reach low limit then trigger fbHomeToSwitch
		    bHomed:=FALSE;
			bSequenceReady:=FALSE;
			fbMoveVelocity.Velocity:=ABS(fbHomePrepare.fVelocityToCam);
            fbMoveVelocity.Direction:=MC_Positive_Direction;
	        bExecuteMoveVelocity:=bExecute;  // Execute MC_MoveVelocity
		    IF NOT bLimitFwd AND NOT fbMoveVelocity.Busy AND Axis.Status.NotMoving THEN //MC_MoveVelocity.Busy goes down when ramp down initiates (not ends).
			  nHomingState:=2;
		    END_IF
		  2: // Wait for fbHomeToSwitch
		    bHomed:=FALSE;
		    bSequenceReady:=FALSE;
            bExecuteMoveVelocity:=FALSE;			
            bExecuteHomeToSwitch:=TRUE;	
            fbHomeToSwitch.nSearchDirTwoardsCam:=MC_Negative_Direction;
            fbHomeToSwitch.nSearchDirOffCam:=MC_Negative_Direction;	             
	        fbHomeToSwitch.fVelocityToCamNC:=fbHomePrepare.fVelocityToCam; // High speed
  	        fbHomeToSwitch.fVelocityFromCamNC:=fbHomePrepare.fVelocityFromCam;  // Low speed              		
		    fbHomeToSwitch.bCamSensor:=bHomeSensor;            	 		    
	        IF fbHomeToSwitch.bDone THEN	          
			  nHomingState:=3;
			  bExecuteFinish:=TRUE;
			  fbHomeFinish.bSofLimEnableHigh:=fbHomePrepare.bSofLimEnableHighOriginal;
			  fbHomeFinish.bSofLimEnableLow:=fbHomePrepare.bSofLimEnableLowOriginal;
	        END_IF;	
          3: // Restore softlimit enable
            bHomed:=FALSE;
		    bSequenceReady:=FALSE;            		            	
	        IF fbHomeFinish.bDone THEN
			  bRestoreNCDataNeeded:=FALSE;
	          bSequenceReady:=TRUE;
			  nHomingState:=0;
			  bHomed:=Axis.Status.Homed;
	        END_IF;	 
	   END_CASE;
		  	    
   15: //Set current position (simplest homing sequence)
     bExecuteHomeDirect:=bExecute;
	 bHomed:=Axis.Status.Homed;
     IF fbHomeDirect.bDone THEN  //Homing ready				
	   bExecuteHomeDirect:=FALSE;				
       bSequenceReady:=TRUE;	
     END_IF	 
	 
ELSE
  fbHomeToSwitch.bCamSensor:=FALSE;
  bHomed:=Axis.Status.Homed;
END_CASE;

// Main homing block
fbHomeToSwitch(
	bExecute:=bExecuteHomeToSwitch AND bExecute AND NOT bError AND NOT bExecuteHomeDirect AND NOT bExecuteMoveVelocity,
 	bReset:=bReset,
	fHomePosition:=fHomePosition,
	Axis:=Axis
);

// Approach limit switch (error if MC_Home is used)
fbMoveVelocity(
    Execute:= bExecuteMoveVelocity AND bExecute AND NOT bError AND NOT bExecuteHomeToSwitch AND NOT bExecuteHomeDirect,
    Axis:=Axis
);

// No sequence, just set position value (nCmdDataLocal=15). Can not run if fbHomeToSwitch is executed
fbHomeDirect(
	bExecute:=bExecuteHomeDirect AND bExecute AND NOT bError  AND NOT bExecuteHomeToSwitch AND NOT bExecuteMoveVelocity,
 	bReset:=bReset,
	fHomePosition:=fHomePosition,
	Axis:=Axis
);

 
//############# Finish homing

IF NOT bexecute AND bRestoreNCDataNeeded THEN  //If homing is aborted restore is needed
	bExecuteFinish:=TRUE;
	IF fbHomeFinish.bDone THEN
	  bExecuteFinish:=FALSE;
      bRestoreNCDataNeeded:=FALSE;	
	END_IF
END_IF

fbHomeFinish(
  En:=En,
  bExecute:=bExecuteFinish,
  bReset:=bReset,
  Axis:=Axis,
);

// Error handling
IF NOT bError THEN
  IF fbHomeToSwitch.bError THEN 
	bError:=fbHomeToSwitch.bError;
	nErrorId:=fbHomeToSwitch.nErrorId;
  ELSIF fbHomeDirect.bError THEN
	bError:=fbHomeDirect.bError;
	nErrorId:=fbHomeDirect.nErrorId;
  ELSIF fbMoveVelocity.Error THEN
	bError:=fbMoveVelocity.Error;
	nErrorId:=fbMoveVelocity.ErrorId;    		    		
  END_IF;	
END_IF

// Done and busy bit
bDone:=bSequenceReady AND bExecute;
bBusy:=NOT bSequenceReady;	 

RETURN;

END_FUNCTION_BLOCK

// tc_mca_std_lib/POUs/Motion/Homing/FB_HomeToSwitch
FUNCTION_BLOCK FB_HomeToSwitch
VAR_INPUT
	En: BOOL;
	bReset: BOOL;
    bExecute: BOOL;	
    bCamSensor:BOOL;	
	nSearchDirTwoardsCam: MC_Direction;
	nSearchDirOffCam: MC_Direction;
	fHomePosition:LREAL;	
	fVelocityToCamNC: LREAL; //Velcoity when searching for cam
	fVelocityFromCamNC: LREAL; // Velocity after found cam (searching for next signal transition)
END_VAR
VAR_IN_OUT
	Axis: AXIS_REF;
END_VAR
VAR_OUTPUT
	EnO: BOOL;	
	bBusy: BOOL;
	bDone: BOOL;
	bHomed:BOOL;
	bError: BOOL;
	nErrorId: UDINT;
END_VAR
VAR
	fbHome: MC_Home;	
	fbWriteHomeDirCamToNC:FB_WriteParameterInNc_v1_00;
	fbWriteHomeDirSyncToNC:FB_WriteParameterInNc_v1_00;
	fbWriteHomeModeToNC:FB_WriteParameterInNc_v1_00;
	fbWriteHomeVelocitiesToNC: FB_HomeWriteNcVelocities;
	bConfigNCDone:BOOL:=FALSE;
	fbRTrigg: R_TRIG;
END_VAR

En:=EnO;
IF bReset THEN
	bConfigNCDone:=FALSE;
	bError:=FALSE;
	nErrorId:=0;
END_IF 
	
//Start preparation of NC if rising edge on bExecute
fbRTrigg(CLK:=bExecute);
IF fbRTrigg.Q THEN
	bConfigNCDone:=FALSE;
END_IF

 
fbWriteHomeDirCamToNC(
	bExecute:=bExecute AND NOT bConfigNCDone,
	nDeviceGroup:=16#5000,
	nIndexOffset:=16#101,	//Direction for Calibration Cam Search	
	nData:=BOOL_TO_DWORD(nSearchDirTwoardsCam=MC_Negative_Direction),//BOOL_TO_DWORD(NOT bSearchDirTwoardsCam),
	Axis:=Axis
);

fbWriteHomeDirSyncToNC(
	bExecute:= bExecute AND NOT bConfigNCDone,
	nDeviceGroup:=16#5000 ,
	nIndexOffset:=16#102 , //Direction for Sync Impuls Search
	nData:=BOOL_TO_DWORD(nSearchDirOffCam=MC_Negative_Direction),//BOOL_TO_DWORD(NOT bSearchDirOffCam),
	Axis:= Axis 
);

fbWriteHomeModeToNC(
	bExecute:=bExecute AND NOT bConfigNCDone,
	nDeviceGroup:=16#5000,
	nIndexOffset:=16#107,  //Reference Mode
	nData:=1,
	Axis:=axis);
	
fbWriteHomeVelocitiesToNC(
  En:=En,
  bExecute:=bExecute AND NOT bConfigNCDone,
  bReset:=bReset,
  fVelocityFromCam:=fVelocityFromCamNC,
  fVelocityToCam:=fVelocityToCamNC,
  Axis:=Axis);

fbHome.bCalibrationCam:=bCamSensor;

fbHome(
	Execute:=bExecute AND bConfigNCDone(* AND NOT bError*),
	Position:=fHomePosition,
	HomingMode:=0,
	Axis:=Axis
	);
bBusy:=(fbHome.Busy OR (NOT bConfigNCDone AND bExecute));
bDone:=fbHome.Done AND bConfigNCDone;
bHomed:=Axis.Status.Homed;

IF (NOT bConfigNCDone) AND fbWriteHomeDirCamToNC.bDone AND fbWriteHomeDirSyncToNC.bDone AND fbWriteHomeModeToNC.bDone AND fbWriteHomeVelocitiesToNC.bDone THEN
  bConfigNCDone:=TRUE;
END_IF

//For some reason MC_HOME gives an Error for one cycle of NC-Task 1 SVB (10ms default..) so filter with bExecute
bError:=(fbHome.Error AND bExecute) OR fbWriteHomeDirCamToNC.bError OR fbWriteHomeDirSyncToNC.bError OR fbWriteHomeModeToNC.bError OR fbWriteHomeVelocitiesToNC.bError;

IF (fbHome.Error AND bExecute) THEN
  nErrorId:=fbHome.ErrorID;
ELSIF fbWriteHomeDirCamToNC.bError THEN
  nErrorId:=fbWriteHomeDirCamToNC.nErrorId;
ELSIF fbWriteHomeDirSyncToNC.bError THEN
  nErrorId:=fbWriteHomeDirSyncToNC.nErrorId;
ELSIF fbWriteHomeModeToNC.bError THEN
  nErrorId:=fbWriteHomeModeToNC.nErrorId;
ELSIF fbWriteHomeVelocitiesToNC.bError THEN
  nErrorId:=fbWriteHomeVelocitiesToNC.nErrorId;  
END_IF

END_FUNCTION_BLOCK

// tc_mca_std_lib/POUs/ChangeConfig/FB_WriteParameterInNc_v1_00
///#########################################################
///Function block to write parameter in Nc.
///
///	Library:		
///	Tc2_MC2.lib
/// Tc2_System.lib
///
///	Global Variables:
///	
///	Data types:
///	
///	External functions:
///
///	History:
///	2014-02-05	v1.00	NB	Release code.
///
///	Known bugs:
///
///
///
///###########################################################
FUNCTION_BLOCK FB_WriteParameterInNc_v1_00
VAR_INPUT
	bExecute: BOOL;
	///16#4000=Axisdata, 16#5000=Encoderdata, 16#6000=Controldata, 16#7000=Drivedata
	nDeviceGroup: UDINT;
	nIndexOffset: UDINT;
	nData: DWORD;
END_VAR
VAR_OUTPUT
	bBusy: BOOL;
	bDone: BOOL;
	bError: BOOL;
	nErrorId: UDINT;
END_VAR
VAR_IN_OUT
	Axis: AXIS_REF;
END_VAR
VAR
	nState: UINT;
	fbADSWRITE: ADSWRITE;
END_VAR

(*Sequence to write parameter in Nc*)
CASE nState OF
0:  (*Start sequence. Wait until bExecute is TRUE*)
	IF bExecute THEN
		bBusy:=TRUE;
		bError:=FALSE;
		nErrorId:=0;
		nState:=10;
	END_IF

10: (*Write parameter in Nc*)
	fbADSWRITE(
		PORT:=500,
		IDXGRP:=nDeviceGroup+Axis.NcToPlc.AxisId,
		IDXOFFS:=nIndexOffset,
		LEN:=SIZEOF(nData),
		SRCADDR:=ADR(nData),
		WRITE:=TRUE);

	(*Wait until it's done or if an error occurs*)
	IF NOT fbADSWRITE.ERR THEN
		IF NOT fbADSWRITE.BUSY THEN
			fbADSWRITE(WRITE:=FALSE);
			nState:=20;
		END_IF
	ELSE
		nErrorId:=fbADSWRITE.ERRID;
		nState:=999;
	END_IF

20: (*Sequense is done. Waits until bExecute is FALSE*)
	bBusy:=FALSE;
	bDone:=TRUE;
	IF NOT bExecute THEN
		bDone:=FALSE;
		nState:=0;
	END_IF

999: (*Error in sequence*)
	bError:=TRUE;
	bBusy:=FALSE;
	bDone:=FALSE;
	fbADSWRITE(WRITE:=FALSE);
	IF NOT bExecute THEN
		nState:=0;
	END_IF

END_CASE

END_FUNCTION_BLOCK

// tc_mca_std_lib/POUs/Motion/Homing/FB_HomeWriteNcVelocities
FUNCTION_BLOCK FB_HomeWriteNcVelocities
VAR_INPUT
	En: BOOL;
	bReset: BOOL;
    bExecute: BOOL;		
	fVelocityToCam: LREAL;
	fVelocityFromCam: LREAL;	
END_VAR
VAR_IN_OUT
	Axis: AXIS_REF;
END_VAR
VAR_OUTPUT
	EnO: BOOL;	
	bBusy: BOOL;
	bDone: BOOL;
	bError: BOOL;
	nErrorId: UDINT;	
END_VAR
VAR
	fbExecuteRiseEdge: R_TRIG;
	fbWriteVelocityToCam:FB_WriteFloatParameter;
	fbWriteVelocityFromCam:FB_WriteFloatParameter;
END_VAR

En:=EnO;
IF bReset THEN
	bError:=FALSE;
	nErrorId:=0;
END_IF 

fbExecuteRiseEdge(CLK:=bExecute);

fbWriteVelocityToCam(
	bExecute:=bExecute,
	nDeviceGroup:= 16#4000,
	nIndexOffset:= 16#6,
	nData:=fVelocityToCam,
	Axis:= Axis);
	
fbWriteVelocityFromCam(
	bExecute:=bExecute,
	nDeviceGroup:= 16#4000,
	nIndexOffset:= 16#7,
	nData:=fVelocityFromCam,
	Axis:= Axis);

bBusy:=fbWriteVelocityFromCam.bBusy OR fbWriteVelocityToCam.bBusy;
bDone:=fbWriteVelocityFromCam.bDone AND fbWriteVelocityToCam.bDone AND bExecute;

bError:=fbWriteVelocityToCam.bError OR fbWriteVelocityFromCam.bError;
IF fbWriteVelocityToCam.bError THEN
  nErrorId:=fbWriteVelocityToCam.nErrorId;
ELSIF fbWriteVelocityFromCam.bError THEN
  nErrorId:=fbWriteVelocityFromCam.nErrorId;
END_IF

END_FUNCTION_BLOCK

// tc_mca_std_lib/POUs/ChangeConfig/FB_WriteFloatParameter
///#########################################################
///Function block to write parameter in Nc.
///
///	Library:		
///	Tc2_MC2.lib
/// Tc2_System.lib
///
///	Global Variables:
///	
///	Data types:
///	
///	External functions:
///
///	History:
///	2014-02-05	v1.00	NB	Release code.
///
///	Known bugs:
///
///
///
///###########################################################
FUNCTION_BLOCK FB_WriteFloatParameter
VAR_INPUT
	bExecute: BOOL;
	///16#4000=Axisdata, 16#5000=Encoderdata, 16#6000=Controldata, 16#7000=Drivedata
	nDeviceGroup: UDINT;
	nIndexOffset: UDINT;
	nData: LREAL;
END_VAR
VAR_OUTPUT
	bBusy: BOOL;
	bDone: BOOL;
	bError: BOOL;
	nErrorId: UDINT;
END_VAR
VAR_IN_OUT
	Axis: AXIS_REF;
END_VAR
VAR
	nState: UINT;
	fbADSWRITE: ADSWRITE;
END_VAR

(*Sequence to write parameter in Nc*)
CASE nState OF
0:  (*Start sequence. Wait until bExecute is TRUE*)
	IF bExecute THEN
		bBusy:=TRUE;
		bError:=FALSE;
		nErrorId:=0;
		nState:=10;
	END_IF

10: (*Write parameter in Nc*)
	fbADSWRITE(
		PORT:=500,
		IDXGRP:=nDeviceGroup+Axis.NcToPlc.AxisId,
		IDXOFFS:=nIndexOffset,
		LEN:=SIZEOF(nData),
		SRCADDR:=ADR(nData),
		WRITE:=TRUE);

	(*Wait until it's done or if an error occurs*)
	IF NOT fbADSWRITE.ERR THEN
		IF NOT fbADSWRITE.BUSY THEN
			fbADSWRITE(WRITE:=FALSE);
			nState:=20;
		END_IF
	ELSE
		nErrorId:=fbADSWRITE.ERRID;
		nState:=999;
	END_IF

20: (*Sequense is done. Waits until bExecute is FALSE*)
	bBusy:=FALSE;
	bDone:=TRUE;
	IF NOT bExecute THEN
		bDone:=FALSE;
		nState:=0;
	END_IF

999: (*Error in sequence*)
	bError:=TRUE;
	bBusy:=FALSE;
	bDone:=FALSE;
	fbADSWRITE(WRITE:=FALSE);
	IF NOT bExecute THEN
		nState:=0;
	END_IF

END_CASE

END_FUNCTION_BLOCK

// tc_mca_std_lib/POUs/Motion/Homing/FB_HomeDirect
FUNCTION_BLOCK FB_HomeDirect
VAR_INPUT
	En: BOOL;
	bReset: BOOL;
    bExecute: BOOL;	
	fHomePosition:LREAL;	
END_VAR
VAR_IN_OUT
	Axis: AXIS_REF;
END_VAR
VAR_OUTPUT
	EnO: BOOL;	
	bBusy: BOOL;
	bDone: BOOL;
	bHomed:BOOL;
	bError: BOOL;
	nErrorId: UDINT;
END_VAR
VAR
	fbHome: MC_Home;	
END_VAR

En:=EnO;
IF bReset THEN
	bError:=FALSE;
	nErrorId:=0;
END_IF 

fbHome(
	Execute:=bExecute,
	Position:=fHomePosition,
	HomingMode:=MC_Direct,
	bCalibrationCam:=FALSE,
	Axis:=Axis
	);
	
bBusy:=fbHome.Busy;
bDone:=fbHome.Done;
bHomed:=Axis.Status.Homed;

bError:=fbHome.Error; 

IF fbHome.Error THEN
  nErrorId:=fbHome.ErrorID;
END_IF

END_FUNCTION_BLOCK

// tc_mca_std_lib/POUs/Motion/Homing/FB_HomePrepare
FUNCTION_BLOCK FB_HomePrepare
VAR_INPUT
	En: BOOL;
	bReset: BOOL;
    bExecute: BOOL;	
    nCmdData: UINT;		
END_VAR
VAR_IN_OUT
	Axis: AXIS_REF;
END_VAR
VAR_OUTPUT
	EnO: BOOL;	
	bBusy: BOOL;
	bDone: BOOL;
	bError: BOOL;
	nErrorId: UDINT;
	bSofLimEnableLowOriginal: BOOL:=TRUE;
	bSofLimEnableHighOriginal: BOOL:=TRUE;	
	fVelocityToCam: LREAL:=0;
	fVelocityFromCam: LREAL:=0;		
END_VAR
VAR
	fbHomeReadSoftLimEnable:FB_HomeReadSoftLimEnable;	
	fbHomeDisableSoftLimEnable:FB_HomeWriteSoftLimEnable;
	fbHomeReadNCVelocities: FB_HomeReadNcVelocities;
	fbHomeResetCalibrationFlag:MC_Home;   //Only used for reset of calibration flag
	fbExecuteRiseEdge: R_TRIG;
	bExecuteReadNC:BOOL:=FALSE;
	bExecuteWriteNC:BOOL:=FALSE;
	nState:INT:=0;
END_VAR

En:=EnO;
IF bReset THEN
	bError:=FALSE;
	nErrorId:=0;
END_IF 

IF NOT bExecute THEN
  bExecuteReadNC:=FALSE;
  bExecuteWriteNC:=FALSE;   
  nState:=0;
END_IF

fbExecuteRiseEdge(CLK:=bExecute);
IF fbExecuteRiseEdge.Q THEN
  bExecuteReadNC:=TRUE;  
END_IF

// Read from NC
fbHomeReadNCVelocities(
  En:=En,
  bExecute:=bExecuteReadNC, // Actualy not needed for sequence 15 (set position only, no movement))
  bReset:=bReset,
  Axis:=Axis,
);

fbHomeReadSoftLimEnable(
	En:=En,
	bExecute:=bExecuteReadNC AND bExecute,
	Axis:=Axis,
	bReset:=bReset,	
);

// Reset calibration flag
fbHomeResetCalibrationFlag(
  Execute:=bExecuteReadNC,
  HomingMode:=MC_ResetCalibration,
  Axis:=Axis
);

bSofLimEnableLowOriginal:=fbHomeReadSoftLimEnable.bSofLimEnableLow;
bSofLimEnableHighOriginal:=fbHomeReadSoftLimEnable.bSofLimEnableHigh;	

fVelocityToCam:=fbHomeReadNCVelocities.fVelocityToCam;
fVelocityFromCam:=fbHomeReadNCVelocities.fVelocityFromCam;

IF bExecuteReadNC AND bExecute AND fbHomeReadSoftLimEnable.bDone THEN
	fbHomeDisableSoftLimEnable.bSofLimEnableHigh:=FALSE;
	fbHomeDisableSoftLimEnable.bSofLimEnableLow:=FALSE;
	bExecuteWriteNC:=TRUE; //Always write (only needed if enabled actually)
END_IF

// Write to NC (disable soft limits)
fbHomeDisableSoftLimEnable(
	En:=En,
	bExecute:=bExecuteWriteNC AND bExecute,
	Axis:=Axis,
	bReset:=bReset,	
);

bBusy:=fbHomeReadSoftLimEnable.bBusy OR fbHomeDisableSoftLimEnable.bBusy OR fbHomeReadNCVelocities.bBusy OR fbHomeResetCalibrationFlag.Busy;
bDone:=fbHomeReadSoftLimEnable.bDone AND fbHomeDisableSoftLimEnable.bDone AND fbHomeReadNCVelocities.bDone AND fbHomeResetCalibrationFlag.Done AND bExecute;

bError:=fbHomeReadSoftLimEnable.bError OR fbHomeDisableSoftLimEnable.bError OR fbHomeReadNCVelocities.bError OR fbHomeResetCalibrationFlag.Error;
IF fbHomeReadSoftLimEnable.bError THEN
  nErrorId:=fbHomeReadSoftLimEnable.nErrorId;
ELSIF fbHomeDisableSoftLimEnable.bError THEN
  nErrorId:=fbHomeDisableSoftLimEnable.nErrorId;
ELSIF fbHomeResetCalibrationFlag.Error THEN
  nErrorId:=fbHomeResetCalibrationFlag.ErrorId;
END_IF

END_FUNCTION_BLOCK

// tc_mca_std_lib/POUs/Motion/Homing/FB_HomeReadSoftLimEnable
FUNCTION_BLOCK FB_HomeReadSoftLimEnable
VAR_INPUT
	En: BOOL;
	bReset: BOOL;
    bExecute: BOOL;			
END_VAR
VAR_IN_OUT
	Axis: AXIS_REF;
END_VAR
VAR_OUTPUT
	EnO: BOOL;	
	bBusy: BOOL;
	bDone: BOOL;
	bError: BOOL;
	nErrorId: UDINT;	
	bSofLimEnableLow: BOOL:=TRUE;
	bSofLimEnableHigh: BOOL:=TRUE;
END_VAR
VAR
	fbReadSoftLimEnableLow:FB_ReadParameterInNc_v1_00;
	fbReadSoftLimEnableHigh:FB_ReadParameterInNc_v1_00;
END_VAR

En:=EnO;
IF bReset THEN
	bError:=FALSE;
	nErrorId:=0;
END_IF 
	
fbReadSoftLimEnableLow(
	bExecute:=bExecute,
	nDeviceGroup:= 16#5000,
	nIndexOffset:= 16#B,
	Axis:= Axis);

fbReadSoftLimEnableHigh(
	bExecute:=bExecute,
	nDeviceGroup:= 16#5000,
	nIndexOffset:= 16#C,
	Axis:= Axis);
	
bSofLimEnableLow:=DWORD_TO_BOOL(fbReadSoftLimEnableLow.nData);
bSofLimEnableHigh:=DWORD_TO_BOOL(fbReadSoftLimEnableHigh.nData);	

bBusy:=fbReadSoftLimEnableLow.bBusy OR fbReadSoftLimEnableHigh.bBusy;
bDone:=fbReadSoftLimEnableLow.bDone AND fbReadSoftLimEnableHigh.bDone AND bExecute;

bError:=fbReadSoftLimEnableLow.bError OR fbReadSoftLimEnableHigh.bError;
IF fbReadSoftLimEnableLow.bError THEN
  nErrorId:=fbReadSoftLimEnableLow.nErrorId;
ELSIF fbReadSoftLimEnableHigh.bError THEN
  nErrorId:=fbReadSoftLimEnableHigh.nErrorId;
END_IF

END_FUNCTION_BLOCK

// tc_mca_std_lib/POUs/ChangeConfig/FB_ReadParameterInNc_v1_00
///#########################################################
///Function block to read parameter in Nc.
///
///	Library:		
///	Tc2_MC2.lib
/// Tc2_System.lib
///
///	Global Variables:
///	
///	Data types:
///	
///	External functions:
///
///	History:
///	2014-02-05	v1.00	NB	Release code.
///
///	Known bugs:
///
///
///
///###########################################################
FUNCTION_BLOCK FB_ReadParameterInNc_v1_00
VAR_INPUT
	bExecute: BOOL;
	///16#4000=Axisdata, 16#5000=Encoderdata, 16#6000=Controldata, 16#7000=Drivedata
	nDeviceGroup: UDINT;
	nIndexOffset: UDINT;
END_VAR
VAR_OUTPUT
	nData: DWORD;
	bBusy: BOOL;
	bDone: BOOL;
	bError: BOOL;
	nErrorId: UDINT;
END_VAR
VAR_IN_OUT
	Axis: AXIS_REF;
END_VAR
VAR
	nState: UINT;
	fbADSREAD: ADSREAD;
END_VAR

(*Sequence to read parameter in Nc*)
CASE nState OF
0:  (*Start sequence. Wait until bExecute is TRUE*)
	IF bExecute THEN
		bBusy:=TRUE;
		bError:=FALSE;
		nErrorId:=0;
		nState:=10;
	END_IF

10: (*Read parameter in Nc*)
	fbADSREAD(
		PORT:=500,
		IDXGRP:=nDeviceGroup+Axis.NcToPlc.AxisId,
		IDXOFFS:=nIndexOffset,
		LEN:=SIZEOF(nData),
		DESTADDR:=ADR(nData),
		READ:=TRUE);

	(*Wait until it's done or if an error occurs*)
	IF NOT fbADSREAD.ERR THEN
		IF NOT fbADSREAD.BUSY THEN
			fbADSREAD(READ:=FALSE);
			nState:=20;
		END_IF
	ELSE
		nErrorId:=fbADSREAD.ERRID;
		nState:=999;
	END_IF

20: (*Sequense is done. Waits until bExecute is FALSE*)
	bBusy:=FALSE;
	bDone:=TRUE;
	IF NOT bExecute THEN
		bDone:=FALSE;
		nState:=0;
	END_IF

999: (*Error in sequence*)
	bError:=TRUE;
	bBusy:=FALSE;
	bDone:=FALSE;
	fbADSREAD(READ:=FALSE);
	IF NOT bExecute THEN
		nState:=0;
	END_IF

END_CASE

END_FUNCTION_BLOCK

// tc_mca_std_lib/POUs/Motion/Homing/FB_HomeWriteSoftLimEnable
FUNCTION_BLOCK FB_HomeWriteSoftLimEnable
VAR_INPUT
	En: BOOL;
	bReset: BOOL;
    bExecute: BOOL;		
	bSofLimEnableLow: BOOL:=TRUE;
	bSofLimEnableHigh: BOOL:=TRUE;
END_VAR
VAR_IN_OUT
	Axis: AXIS_REF;
END_VAR
VAR_OUTPUT
	EnO: BOOL;	
	bBusy: BOOL;
	bDone: BOOL;
	bError: BOOL;
	nErrorId: UDINT;	
END_VAR
VAR
	fbExecuteRiseEdge: R_TRIG;
	fbWriteSoftLimEnableLow:FB_WriteParameterInNc_v1_00;
	fbWriteSoftLimEnableHigh:FB_WriteParameterInNc_v1_00;
END_VAR

En:=EnO;
IF bReset THEN
	bError:=FALSE;
	nErrorId:=0;
END_IF 

fbExecuteRiseEdge(CLK:=bExecute);

fbWriteSoftLimEnableLow(
	bExecute:=bExecute,
	nDeviceGroup:= 16#5000,
	nIndexOffset:= 16#B,
	nData:=BOOL_TO_DWORD(bSofLimEnableLow),
	Axis:= Axis);
	
fbWriteSoftLimEnableHigh(
	bExecute:=bExecute,
	nDeviceGroup:= 16#5000,
	nIndexOffset:= 16#C,
	nData:=BOOL_TO_DWORD(bSofLimEnableHigh),
	Axis:= Axis);

bBusy:=fbWriteSoftLimEnableLow.bBusy OR fbWriteSoftLimEnableHigh.bBusy;
bDone:=fbWriteSoftLimEnableLow.bDone AND fbWriteSoftLimEnableHigh.bDone AND bExecute;

bError:=fbWriteSoftLimEnableHigh.bError OR fbWriteSoftLimEnableLow.bError;
IF fbWriteSoftLimEnableHigh.bError THEN
  nErrorId:=fbWriteSoftLimEnableHigh.nErrorId;
ELSIF fbWriteSoftLimEnableLow.bError THEN
  nErrorId:=fbWriteSoftLimEnableLow.nErrorId;
END_IF

END_FUNCTION_BLOCK

// tc_mca_std_lib/POUs/Motion/Homing/FB_HomeReadNcVelocities
FUNCTION_BLOCK FB_HomeReadNcVelocities
VAR_INPUT
	En: BOOL;
	bReset: BOOL;
    bExecute: BOOL;			
END_VAR
VAR_IN_OUT
	Axis: AXIS_REF;
END_VAR
VAR_OUTPUT
	EnO: BOOL;	
	bBusy: BOOL;
	bDone: BOOL;
	bError: BOOL;
	nErrorId: UDINT;	
	fVelocityToCam: LREAL;
	fVelocityFromCam: LREAL;
END_VAR
VAR
	fbReadVelocityToCam:FB_ReadFloatParameter;
	fbReadVelocityFromCam:FB_ReadFloatParameter;
END_VAR

En:=EnO;
IF bReset THEN
	bError:=FALSE;
	nErrorId:=0;
END_IF 
	
fbReadVelocityToCam(
	bExecute:=bExecute,
	nDeviceGroup:= 16#4000,
	nIndexOffset:= 16#6,
	Axis:= Axis);
	
fbReadVelocityFromCam(
	bExecute:=bExecute,
	nDeviceGroup:= 16#4000,
	nIndexOffset:= 16#7,
	Axis:= Axis);
	
fVelocityToCam:=fbReadVelocityToCam.nData;
fVelocityFromCam:=fbReadVelocityFromCam.nData;	

bBusy:=fbReadVelocityFromCam.bBusy OR fbReadVelocityToCam.bBusy;
bDone:=fbReadVelocityFromCam.bDone AND fbReadVelocityToCam.bDone AND bExecute;

bError:=fbReadVelocityToCam.bError OR fbReadVelocityFromCam.bError;
IF fbReadVelocityToCam.bError THEN
  nErrorId:=fbReadVelocityToCam.nErrorId;
ELSIF fbReadVelocityFromCam.bError THEN
  nErrorId:=fbReadVelocityFromCam.nErrorId;
END_IF

END_FUNCTION_BLOCK

// tc_mca_std_lib/POUs/ChangeConfig/FB_ReadFloatParameter
FUNCTION_BLOCK FB_ReadFloatParameter
VAR_INPUT
	bExecute: BOOL;
	///16#4000=Axisdata, 16#5000=Encoderdata, 16#6000=Controldata, 16#7000=Drivedata
	nDeviceGroup: UDINT;
	nIndexOffset: UDINT;
END_VAR
VAR_OUTPUT
	nData: LREAL;
	bBusy: BOOL;
	bDone: BOOL;
	bError: BOOL;
	nErrorId: UDINT;
END_VAR
VAR_IN_OUT
	Axis: AXIS_REF;
END_VAR
VAR
	nState: UINT;
	fbADSREAD: ADSREAD;
END_VAR

(*Sequence to read parameter in Nc*)
CASE nState OF
0:  (*Start sequence. Wait until bExecute is TRUE*)
	IF bExecute THEN
		bBusy:=TRUE;
		bError:=FALSE;
		nErrorId:=0;
		nState:=10;
	END_IF

10: (*Read parameter in Nc*)
	fbADSREAD(
		PORT:=500,
		IDXGRP:=nDeviceGroup+Axis.NcToPlc.AxisId,
		IDXOFFS:=nIndexOffset,
		LEN:=SIZEOF(nData),
		DESTADDR:=ADR(nData),
		READ:=TRUE);

	(*Wait until it's done or if an error occurs*)
	IF NOT fbADSREAD.ERR THEN
		IF NOT fbADSREAD.BUSY THEN
			fbADSREAD(READ:=FALSE);
			nState:=20;
		END_IF
	ELSE
		nErrorId:=fbADSREAD.ERRID;
		nState:=999;
	END_IF

20: (*Sequense is done. Waits until bExecute is FALSE*)
	bBusy:=FALSE;
	bDone:=TRUE;
	IF NOT bExecute THEN
		bDone:=FALSE;
		nState:=0;
	END_IF

999: (*Error in sequence*)
	bError:=TRUE;
	bBusy:=FALSE;
	bDone:=FALSE;
	fbADSREAD(READ:=FALSE);
	IF NOT bExecute THEN
		nState:=0;
	END_IF

END_CASE

END_FUNCTION_BLOCK

// tc_mca_std_lib/POUs/Motion/Homing/FB_HomeFinish
FUNCTION_BLOCK FB_HomeFinish
VAR_INPUT
	En: BOOL;
	bReset: BOOL;
    bExecute: BOOL;	
    nCmdData: UINT;
	bSofLimEnableLow: BOOL:=TRUE;
	bSofLimEnableHigh: BOOL:=TRUE;			
END_VAR
VAR_IN_OUT
	Axis: AXIS_REF;
END_VAR
VAR_OUTPUT
	EnO: BOOL;	
	bBusy: BOOL;
	bDone: BOOL;
	bError: BOOL;
	nErrorId: UDINT;
END_VAR
VAR		
	fbHomewriteSoftLimEnable:FB_HomeWriteSoftLimEnable;	
	fbExecuteRiseEdge: R_TRIG;	
	bExecuteWriteNC:BOOL:=FALSE;
	nState:INT:=0;
END_VAR

En:=EnO;
IF bReset THEN
	bError:=FALSE;
	nErrorId:=0;
END_IF 

IF NOT bExecute THEN
  bExecuteWriteNC:=FALSE;
  fbHomewriteSoftLimEnable.bSofLimEnableLow:=bSofLimEnableLow;
  fbHomewriteSoftLimEnable.bSofLimEnableHigh:=bSofLimEnableHigh;   
  nState:=0;
END_IF

fbExecuteRiseEdge(CLK:=bExecute);
IF fbExecuteRiseEdge.Q THEN
  bExecuteWriteNC:=TRUE;  
  fbHomewriteSoftLimEnable.bSofLimEnableLow:=bSofLimEnableLow;
  fbHomewriteSoftLimEnable.bSofLimEnableHigh:=bSofLimEnableHigh;
END_IF

// Write to NC (disable soft limits)
fbHomewriteSoftLimEnable(
	En:=En,
	bExecute:=bExecuteWriteNC AND bExecute,
	Axis:=Axis,
	bReset:=bReset,	
);

bBusy:=fbHomewriteSoftLimEnable.bBusy;
bDone:=fbHomewriteSoftLimEnable.bDone;

bError:=fbHomewriteSoftLimEnable.bError;
IF fbHomewriteSoftLimEnable.bError THEN
  nErrorId:=fbHomewriteSoftLimEnable.nErrorId;
END_IF

END_FUNCTION_BLOCK

// POUs/Motion/Utils/FB_SetEnables
FUNCTION_BLOCK FB_SetEnables
// Update the all enable booleans based on the booleans that make them up
VAR_IN_OUT
    stMotionStage: DUT_MotionStage;
END_VAR

stMotionStage.bAllForwardEnable := stMotionStage.bLimitForwardEnable AND (stMotionStage.bGantryForwardEnable OR NOT stMotionStage.bGantryAxis);
stMotionStage.bAllBackwardEnable := stMotionStage.bLimitBackwardEnable AND (stMotionStage.bGantryBackwardEnable OR NOT stMotionStage.bGantryAxis);

stMotionStage.bAllEnable := stMotionStage.bEnable AND stMotionStage.bHardwareEnable;

END_FUNCTION_BLOCK

// POUs/Motion/FB_EncoderValue
FUNCTION_BLOCK FB_EncoderValue
(*
    Process the encoder value for DUT_MotionStage

    A few different problems this is trying to solve:
        1. Different encoders show as different types in the IO,
           but we want a consistent type for checks and for PVs
        2. Some inverted encoders display as very high numbers
           as they count down from max int instead of up from 0
        3. Some encoders have raw signed values, others unsigned.

    To this end, we figure out which encoder is linked and process
    the value appropriately.
*)
VAR_IN_OUT
    stMotionStage: DUT_MotionStage;
END_VAR

IF stMotionStage.nRawEncoderULINT <> 0 THEN
    IF stMotionStage.nRawEncoderULINT < 4294967296 THEN
        stMotionStage.nEncoderCount := ULINT_TO_UDINT(stMotionStage.nRawEncoderULINT);
    ELSE
        stMotionStage.nEncoderCount := ULINT_TO_UDINT(18446744073709551615 - stMotionStage.nRawEncoderULINT);
    END_IF
ELSIF stMotionStage.nRawEncoderUINT <> 0 THEN
    stMotionStage.nEncoderCount := UINT_TO_UDINT(stMotionStage.nRawEncoderUINT);
ELSIF stMotionStage.nRawEncoderINT <> 0 THEN
    stMotionStage.nEncoderCount := INT_TO_UDINT(stMotionStage.nRawEncoderINT);
ELSE
    stMotionStage.nEncoderCount := 0;
END_IF

END_FUNCTION_BLOCK

// POUs/Motion/FB_MotionStageNCParams
FUNCTION_BLOCK FB_MotionStageNCParams
(*
    Read and refresh axis parameters struct on DUT_MotionStage
*)
VAR_IN_OUT
    stMotionStage: DUT_MotionStage;
END_VAR
VAR_INPUT
    bEnable: BOOL;
    tRefreshDelay: TIME;
END_VAR
VAR_OUTPUT
    bError: BOOL;
END_VAR
VAR
    mcReadParams: MC_ReadParameterSet;
    timer: TON;
    bExecute: BOOL := TRUE;
    nLatchErrId: UDINT;
END_VAR

